Yaskawa INFORM job: OK_R2_O57-69(1)(90,0)_OK.JBI

/JOB
//NAME OK_R2_O57-69(1)(90,0)_OK
///FOLDERNAME X4
//POS
///NPOS 455,455,455,17,0,0
///TOOL 0
///POSTYPE PULSE
///PULSE
C00000=142687,-11580,-21865,-46298,77318,26406
C00001=107635,105639,59193,-4004,83878,4369
C00002=107385,112835,71659,-3962,79901,4413
C00003=107289,116273,78306,-3960,77580,4454
C00004=107289,116207,79332,-3970,76915,4475
C00005=107289,116273,78306,-3960,77580,4454
C00006=107447,123392,87902,-4042,75345,4582
C00007=107368,119615,82796,-3999,76540,4514
C00008=107503,109882,68607,-3993,80266,4441
C00009=107756,103001,56611,-4038,84116,4400
C00010=108153,102502,65455,-9976,80197,11407
C00011=107537,110693,79141,-9943,75970,11537
C00012=107296,115242,87458,-9996,73200,11681
C00013=107296,115607,88878,-10031,72523,11737
C00014=107296,115242,87458,-9996,73200,11681
C00015=106873,122679,97490,-10001,70830,11727
C00016=107051,118089,91280,-9973,72293,11668
C00017=107734,107812,76377,-9988,76211,11587
C00018=108357,99970,63216,-10030,80298,11469
C00019=111395,81814,40298,-10763,85374,12058
C00020=135939,40633,60147,-39777,44722,28223
C00021=135273,44440,65799,-40560,43252,28620
C00022=135218,49510,74479,-42532,41149,29811
C00023=135218,52739,80290,-44069,39733,30719
C00024=135218,51401,77909,-43430,40304,30344
C00025=135400,47409,73389,-42907,40927,30065
C00026=135400,49581,77316,-43951,39968,30683
C00027=135083,52398,80539,-44303,39430,30833
C00028=135400,49581,77316,-43951,39968,30683
C00029=133089,26435,31840,-33362,51762,23582
C00030=122836,-20707,-1842,-26261,58142,44331
C00031=108542,-11029,1672,-9630,61367,37079
C00032=108679,-9299,6685,-9878,59219,37321
C00033=108679,-8233,9358,-9991,58138,37420
C00034=108679,-8832,7868,-9928,58739,37363
C00035=101227,-4424,8478,6098,64645,33408
C00036=101749,-3909,10367,6019,63714,33552
C00037=99890,-2844,11238,6455,63869,32869
C00038=101954,-4018,10279,5971,63698,33629
C00039=119599,-21935,-8687,-19541,65328,41245
C00040=157787,18659,24844,-603,57771,19260
C00041=142866,15340,32539,5422,51765,13080
C00042=142866,17061,36428,5538,50265,12998
C00043=142866,16346,34832,5489,50877,13033
C00044=143013,20262,38513,5445,50617,13080
C00045=142866,16346,34832,5489,50877,13033
C00046=132913,34622,53415,24401,61187,-11407
C00047=133468,34916,53719,24326,60995,-11227
C00048=131729,29112,41902,23735,65422,-10932
C00049=97397,-56372,-66081,25937,96155,-17363
C00050=91007,-59958,-65967,24261,97668,-32617
C00051=125926,-77250,-66316,21080,81833,-36437
C00052=126284,-594,-20029,15604,88354,-35723
C00053=126284,-509,-12976,15645,84209,-36248
C00054=124802,3877,-7879,15893,83645,-36839
C00055=124802,4020,-6552,15911,82926,-36931
C00056=124802,3943,-7243,15902,83298,-36884
C00057=123270,3785,-7378,16131,83600,-37383
C00058=123399,3884,-6575,16123,83149,-37397
C00059=123813,3922,-6544,16060,83068,-37263
C00060=123399,3797,-7355,16113,83568,-37342
C00061=129363,-46213,-49135,15183,82438,-35396
C00062=131818,-93939,-91511,4308,83147,-7603
C00063=129147,-104974,-80844,-32439,31226,48978
C00064=127581,-72421,-62371,-35585,33961,68342
C00065=124664,-66928,-57448,-32966,32611,66961
C00066=123754,-63943,-53853,-32629,31684,66786
C00067=123754,-63568,-52544,-33171,31167,67071
C00068=123754,-63943,-53853,-32629,31684,66786
C00069=123639,-59018,-51277,-31710,32448,66301
C00070=123582,-56512,-49922,-31282,32817,66076
C00071=123639,-59018,-51277,-31710,32448,66301
C00072=131982,-55244,-47165,-50372,40396,73195
C00073=130304,-55630,-47379,-49442,39430,72657
C00074=124207,-63622,-54438,-32639,32305,66790
C00075=125315,-65804,-56448,-33641,32835,67317
C00076=128233,-71228,-61365,-36187,34229,68662
C00077=123372,-90110,-48954,-69127,12132,-32175
C00078=164723,-27709,-11098,-69634,69545,-47097
C00079=168592,-14054,-1264,-69323,72507,-47019
C00080=158796,970,10778,-68977,66045,-48502
C00081=178190,-60094,-55002,-67962,82251,-43615
C00082=173027,-67602,-58858,-67784,78202,-43687
C00083=169341,-70270,-58661,-67804,75132,-43553
C00084=169341,-69900,-57436,-67934,74906,-43308
C00085=169341,-70270,-58661,-67804,75132,-43553
C00086=168190,-69795,-58431,-67693,74405,-43758
C00087=166974,-69170,-58127,-67562,73648,-43988
C00088=168190,-69795,-58431,-67693,74405,-43758
C00089=173339,-68324,-59217,-67832,78352,-43578
C00090=179024,-58740,-54280,-67998,82909,-43609
C00091=180089,-62311,-56169,-68129,83355,-43176
C00092=195989,-67260,-58691,-68544,93647,-40636
C00093=215727,-82846,-65910,-66533,105415,-36335
C00094=205418,-117613,-84907,-62264,88933,-23433
C00095=200540,-66438,-67217,-63628,100285,15829
C00096=127293,-88890,-117674,-21964,112183,47373
C00097=127884,-113870,-117586,-20406,100261,49782
C00098=126455,-94233,-83658,-19548,96625,49926
C00099=122769,-95152,-80887,-19686,93685,49072
C00100=121257,-92855,-76623,-19731,91957,48808
C00101=121256,-92184,-75240,-19721,91480,48885
C00102=121257,-92855,-76623,-19731,91957,48808
C00103=119709,-92847,-76620,-19813,91585,48312
C00104=118447,-92805,-76604,-19874,91287,47906
C00105=121134,-93057,-78029,-19757,92646,48652
C00106=122616,-92853,-79205,-19699,93786,49000
C00107=126246,-91944,-81970,-19569,96706,49837
C00108=116739,-91029,-87152,11175,94833,-69838
C00109=118638,-93558,-84500,11112,91693,-69464
C00110=121559,-94813,-81066,11067,88585,-68734
C00111=121559,-94454,-79960,11067,88097,-68778
C00112=121559,-94813,-81066,11067,88585,-68734
C00113=121580,-97932,-82261,11067,87731,-68801
C00114=121559,-94813,-81066,11067,88585,-68734
C00115=124478,-94674,-81011,11026,88221,-67759
C00116=121559,-94813,-81066,11067,88585,-68734
C00117=121199,-93273,-83309,11082,90766,-68663
C00118=119237,-90980,-86060,11143,93854,-69064
C00119=119262,-91078,-98551,11400,101347,-68370
C00120=119262,-88450,-105465,11733,106843,-67839
C00121=123634,-129086,-124562,-18007,62786,21453
C00122=124713,-112307,-109989,-18584,62695,21889
C00123=121750,-102661,-104576,-16897,63614,20597
C00124=120661,-96847,-100545,-16291,63882,20142
C00125=120661,-96945,-99213,-16408,63045,20264
C00126=120661,-96847,-100545,-16291,63882,20142
C00127=119434,-96825,-100537,-15680,63651,19709
C00128=118199,-96764,-100511,-15059,63439,19270
C00129=119434,-96825,-100537,-15680,63651,19709
C00130=120468,-95018,-99831,-16130,64325,20004
C00131=120473,-92385,-98782,-16042,65005,19908
C00132=120468,-95018,-99831,-16130,64325,20004
C00133=121400,-102567,-103315,-16828,62845,20579
C00134=124338,-112119,-108698,-18515,61948,21869
C00135=115152,-110094,-108973,21966,66789,-27187
C00136=118701,-101887,-103909,20282,66922,-25804
C00137=120033,-96498,-99821,19662,66842,-25314
C00138=120033,-96571,-98630,19770,66116,-25442
C00139=120033,-96498,-99821,19662,66842,-25314
C00140=121038,-96503,-99823,19217,66607,-24975
C00141=122863,-96447,-99800,18396,66209,-24352
C00142=121038,-96503,-99823,19217,66607,-24975
C00143=121031,-93073,-98698,19079,67622,-24806
C00144=121028,-91162,-97925,19016,68103,-24728
C00145=121031,-93073,-98698,19079,67622,-24806
C00146=119849,-101075,-102503,19842,66224,-25492
C00147=116381,-109262,-107580,21511,66068,-26853
C00148=114174,-113759,-109466,25218,61256,-29915
C00149=117999,-105066,-104585,23039,61495,-28291
C00150=119436,-99712,-100384,22286,61259,-27759
C00151=119436,-99710,-99356,22420,60673,-27881
C00152=119436,-99712,-100384,22286,61259,-27759
C00153=121229,-99730,-100389,21374,60785,-27131
C00154=123455,-99637,-100354,20211,60254,-26337
C00155=121229,-99730,-100389,21374,60785,-27131
C00156=121193,-87849,-97584,20616,64895,-26352
C00157=121184,-85182,-96456,20515,65531,-26236
C00158=121193,-87849,-97584,20616,64895,-26352
C00159=119818,-94456,-100985,21520,64018,-27049
C00160=116346,-102514,-105912,23431,63914,-28430
C00161=120616,-96535,-104175,23887,64719,-45568
C00162=120616,-96992,-102054,24182,63306,-45881
C00163=136389,-91621,-102582,2930,64785,-40204
C00164=118869,-97062,-101163,25162,63282,-46587
C00165=120614,-98220,-102778,24220,63138,-45920
C00166=133621,-94767,-111832,11795,91375,-37411
C00167=135524,-95930,-105043,10399,87493,-38783
C00168=135817,-95923,-103691,10152,86855,-39072
C00169=120616,-96793,-103087,23408,87451,-42960
C00170=120617,-96070,-105685,23410,89266,-42604
C00171=120635,-118119,-124325,17957,114364,-37370
C00172=107148,-122068,-106720,37591,45003,-56343
C00173=107143,-118125,-97071,40168,41922,-57944
C00174=107140,-117153,-94914,40772,41285,-58308
C00175=108973,-111199,-92224,38587,41539,-56980
C00176=105115,-116142,-93852,42098,42144,-59139
C00177=107012,-118507,-95796,40965,41228,-58425
C00178=106841,-125065,-112650,27659,77705,-49700
C00179=108922,-124444,-112086,25532,82947,-48175
C00180=119544,-112769,-109618,11884,115103,-48129
C00181=107149,-124464,-114807,14035,115464,-42498
C00182=107153,-124980,-118069,14274,117155,-42276
C00183=120683,-72727,-118704,1403,106780,-1205
C00184=120616,-97084,-101761,-23685,56760,46645
C00185=120615,-97341,-97713,-24403,54354,47226
C00186=120615,-97245,-95574,-24781,53197,47519
C00187=114204,-97094,-94072,-16119,48782,41960
C00188=120613,-98403,-96349,-24817,53089,47545
C00189=122362,-97151,-94697,-25998,53280,48291
C00190=118994,-95787,-106265,-23004,89078,41795
C00191=118527,-107245,-109313,-22939,85243,42364
C00192=120617,-95328,-107797,-23350,90604,42068
C00193=120618,-93989,-110172,-23402,92584,41681
C00194=120619,-87370,-116055,-23793,99045,40394
C00195=120619,-87370,-116055,-23793,99045,40394
C00196=120618,-86394,-114990,8935,74593,77376
C00197=120618,-89943,-112390,9089,71210,77123
C00198=120618,-91094,-111253,9157,69935,77026
C00199=120921,-87010,-110025,8929,71231,77225
C00200=120616,-91696,-112687,9127,70502,77069
C00201=120617,-91433,-110915,9280,69085,76949
C00202=120617,-91707,-110620,9342,68290,76888
C00203=120617,-92092,-110153,9289,66860,76810
C00204=120617,-92703,-109346,8604,64312,76688
C00205=120617,-93084,-108807,7222,62458,76641
C00206=120617,-93193,-108666,5837,61715,76664
C00207=120618,-90875,-111661,5103,64613,76670
C00208=120618,-90809,-111742,4197,64653,76687
C00209=120618,-90545,-112027,2634,65244,76730
C00210=120618,-90001,-112556,1051,66686,76779
C00211=120618,-89211,-113241,-130,68806,76818
C00212=120618,-88484,-113805,-667,70701,76840
C00213=120618,-87123,-114601,-725,72803,76709
C00214=120619,-86169,-115177,-666,75079,76754
C00215=120619,-85009,-115798,44,77805,76866
C00216=120619,-84186,-116189,1368,79788,77043
C00217=120619,-83945,-116287,2643,80551,77203
C00218=118270,-87908,-113898,4548,77310,76315
C00219=117006,-87882,-113777,5977,77383,75992
C00220=115001,-87936,-113393,8376,77055,75464
C00221=113157,-88199,-112730,10795,75966,74930
C00222=112003,-88721,-111920,12625,74164,74513
C00223=111959,-89151,-111512,13141,72976,74431
C00224=114352,-90005,-111461,12180,71784,75105
C00225=117604,-90791,-111341,10710,70486,76060
C00226=117404,-89600,-112462,10735,71791,76111
C00227=116906,-85938,-115017,10812,75246,76259
C00228=120614,-97623,-100799,20300,88883,-51757
C00229=120614,-96302,-87355,20440,81742,-52958
C00230=120613,-95405,-83784,20521,80111,-53236
C00231=126109,-109592,-85843,18017,65653,-40663
C00232=119108,-93712,-82042,20736,80300,-53753
C00233=120703,-96440,-84059,20528,79748,-53266
C00234=121011,-95101,-82657,16234,85393,-56932
C00235=120815,-94676,-79544,16280,83804,-57215
C00236=120149,-97496,-80464,13581,88226,-67082
C00237=120613,-95181,-82964,13310,91650,-67966
C00238=120614,-96223,-86939,13345,93512,-67766
C00239=120615,-97634,-95801,13498,98116,-67263
C00240=121294,-114205,-91205,-24827,58618,34956
C00241=120612,-94063,-79189,-30374,49118,27390
C00242=120612,-92317,-74276,-31337,47279,28045
C00243=120611,-91635,-72532,-31685,46659,28276
C00244=118073,-86207,-69815,-27979,45725,25770
C00245=120609,-92794,-73597,-31655,46709,28256
C00246=122365,-91337,-71823,-32796,47086,29053
C00247=115372,-110415,-90260,-20403,67055,37755
C00248=116442,-100471,-77078,-21305,66259,40654
C00249=116372,-94168,-76064,-20320,81539,56413
C00250=120612,-93792,-78416,-23522,88402,60481
C00251=120613,-94966,-82014,-23532,89885,60189
C00252=192979,-49879,-84133,-31949,90821,59300
C00253=226136,-49296,-77583,-43048,96139,60221
C00254=194231,-43574,-37464,-64429,96533,-35524
C00255=168190,-921,2356,-69742,86936,-65420
C00256=167171,-9679,-4727,-69794,80481,-66551
C00257=161668,-12899,-4972,-71887,72051,-48991
C00258=158364,-12022,-5998,-68672,69294,-39906
C00259=156881,-17849,-10944,-69825,79076,-66625
C00260=156054,-17027,-11609,-69675,78824,-67093
C00261=158331,-12175,-6115,-68672,69269,-39907
C00262=156361,-14598,-7677,-68484,66767,-40276
C00263=151900,-18330,-10475,-67308,59054,-41902
C00264=154261,3537,6976,-69079,75732,-38618
C00265=154747,-10639,-6391,-66828,75297,-54318
C00266=154442,-11587,-10980,-61883,80878,-64503
C00267=159305,-13086,-7363,-68622,70046,-39902
C00268=160610,-11568,-6196,-68690,70948,-39749
C00269=179726,-19719,-12316,-69264,83687,-37039
C00270=180202,-65513,-36112,-70171,79517,-38597
C00271=171321,-47804,-23743,-70196,73038,-45095
C00272=120855,-117042,-83065,-287,50429,281
C00273=120852,-56541,-79529,-233,79340,219
C00274=120696,53119,40617,-185,61751,192
C00275=120686,117420,104140,-194,55702,198
C00276=120685,99043,82380,-184,59649,191
C00277=122493,102932,90070,-987,56926,916
C00278=120685,123863,115449,-202,52052,205
C00279=120704,115543,105340,-205,53998,209
C00280=122467,102927,90062,-975,56928,906
C00281=121054,101096,87697,-350,57430,341
C00282=121218,100526,86952,-2924,57717,2680
C00283=119871,97554,82980,-2313,58589,2128
C00284=121770,99804,85898,-7979,58802,7335
C00285=123458,93230,74100,-8365,62819,7694
C00286=127901,89142,85055,-16058,61001,15638
C00287=140740,128608,122591,-17053,51761,14935
C00288=141173,120915,113217,-16837,53591,14809
C00289=125539,79311,72650,-14999,63041,14428
C00290=124982,76834,69616,-14757,63515,14150
C00291=126480,71694,61185,-14909,66256,14364
C00292=127425,72489,65068,-16510,65063,16091
C00293=151716,35869,40711,-43800,85634,42977
C00294=153219,23704,46468,-39932,89274,45297
C00295=150010,47902,71614,-40707,85512,45394
C00296=154240,23283,29848,-40334,97498,42612
C00297=154465,34676,28167,-3963,80968,257
C00298=157399,18456,15561,6305,73633,-11364
C00299=166913,17393,14571,4349,73064,-8034
C00300=170742,26415,26762,1268,69531,-3078
C00301=170212,26486,27746,1388,68971,-3275
C00302=169116,27159,30341,1645,67741,-3687
C00303=176334,39723,42022,-11916,74582,1979
C00304=182119,52793,59875,-23973,76306,25334
C00305=185046,47030,49277,-23757,80416,25586
C00306=156159,-27844,-33931,-20967,84276,14245
C00307=135002,-107739,-89418,-17788,72722,8424
C00308=182779,-47107,-63468,-4299,76483,-82831
C00309=189334,-126614,-108463,-44477,62316,-64668
C00310=121693,-126430,-88761,-53982,17457,-73114
C00311=140282,-82155,-73154,-59383,46557,-69401
C00312=137402,-83281,-73645,-58395,44635,-69973
C00313=132931,-76557,-73113,-49425,46479,-74892
C00314=136898,-85885,-74084,-59112,43749,-69513
C00315=136236,-83853,-74475,-57682,44042,-70397
C00316=132981,-76543,-73106,-49450,46508,-74878
C00317=119425,-90003,-77331,-28870,26914,-75911
C00318=135712,-71182,-68173,-46953,38713,-58640
C00319=143905,-59721,-61352,-57730,51418,-39205
C00320=121775,-86236,-74909,-25532,24619,-52498
C00321=121774,-86244,-74912,-25532,24617,-52498
C00322=121693,-126430,-88761,-53982,17457,-73114
C00323=118534,-85327,-101542,31688,82312,-3081
C00324=113867,24354,-27186,33136,92965,-1727
C00325=160796,40344,30640,17217,54638,7315
C00326=160797,40341,30637,17217,54638,7315
C00327=160797,40341,30637,17217,54638,7315
C00328=160252,39151,28676,17378,55324,7200
C00329=161178,38223,28434,16963,54814,7508
C00330=160796,40350,30646,17218,54637,7315
C00331=160795,40351,30648,17218,54637,7314
C00332=160794,40354,30651,17218,54637,7314
C00333=134054,6396,-12292,27269,70214,-305
C00334=134055,6392,-12295,27269,70214,-305
C00335=134055,6392,-12295,27269,70214,-305
C00336=133335,6117,-13247,27465,70843,-432
C00337=134208,4264,-14132,27207,70198,-248
C00338=134055,6400,-12288,27269,70214,-305
C00339=134054,6402,-12286,27269,70214,-305
C00340=134054,6405,-12283,27270,70214,-305
C00341=134054,6378,-12307,27269,70215,-305
C00342=110297,92470,61471,162,75039,5870
C00343=106536,92878,46535,-6489,85409,6991
C00344=105889,102407,60005,-6334,81981,6955
C00345=107411,109724,75819,-6896,76174,7779
C00346=107307,113841,80039,-6878,75687,7770
C00347=106147,102899,60646,-6410,81858,7045
C00348=107454,121313,92229,795,70933,3205
C00349=107823,121162,91899,673,71054,3335
C00350=103297,112702,80407,10779,76295,-8281
C00351=100760,114985,83493,16597,79533,-16127
C00352=102994,101893,66401,15964,82735,-14918
C00353=102438,121053,88749,15854,82872,-18908
C00354=103348,86539,46576,12183,80201,-18226
C00355=107306,113906,81371,827,73803,3171
C00356=107311,117545,72428,-13995,85411,11857
C00357=105409,119135,76795,-9100,84379,11874
C00358=104759,108123,65686,-7737,79041,12181
C00359=107310,116811,74228,-14018,83968,12019
C00360=107566,113040,70432,-14074,84397,12057
C00361=105955,98232,55061,-11625,77681,12450
C00362=106075,100097,56813,-12565,79285,12270
C00363=104774,97118,52951,-12100,79924,11770
C00364=104167,97049,52732,-11892,79935,11566
C00365=103488,98146,54277,-11675,79461,11386
C00366=105019,93844,46472,-12276,82982,11528
C00367=107312,117616,72525,-13996,85389,11860
C00368=113054,94415,53645,-15341,86201,13636
C00369=132655,10139,3212,-19793,78564,21692
C00370=120395,-86682,-93138,-17072,84894,16376
C00371=120731,-81008,-115648,105,86416,81801
C00372=120675,-24654,-47163,132,73228,81771
C00373=120676,-24640,-47153,131,73229,81771
C00374=121102,-22780,-44290,-48,72423,81914
C00375=120676,-24370,-48215,131,74021,81772
C00376=121750,-24626,-47144,-317,73232,82133
C00377=121088,-18910,-41523,-41,72708,81911
C00378=120676,-24640,-47153,131,73229,81771
C00379=120672,-32524,-49889,133,70864,81769
C00380=86683,-40445,-63075,13763,77736,70672
C00381=103499,26970,-9106,7161,77072,76192
C00382=140778,108078,66600,20509,92089,48724
C00383=140778,108101,66629,20508,92083,48723
C00384=140777,108123,66659,20508,92077,48722
C00385=140791,110557,71328,20474,90549,48468
C00386=140777,108420,65802,20527,92715,48830
C00387=141368,109052,67884,20414,91674,48860
C00388=140538,117676,80864,20492,88534,48038
C00389=140777,108123,66659,20508,92077,48722
C00390=140778,108101,66629,20508,92083,48723
C00391=140778,108101,66629,20508,92083,48723
C00392=140778,108122,66658,20508,92077,48722
C00393=140768,108703,68758,20489,91145,48562
C00394=140777,108420,65801,20527,92715,48830
C00395=141368,109051,67883,20414,91674,48860
C00396=140511,115176,77354,20500,89363,48171
C00397=140778,108122,66658,20508,92077,48722
C00398=140778,108100,66628,20508,92083,48723
C00399=140778,108078,66599,20509,92089,48724
C00400=126581,14025,-47477,25241,115824,48542
C00401=159492,92702,46653,29136,105568,44545
C00402=162149,88036,41181,28914,105145,45798
C00403=163325,88052,47564,28312,101300,45262
C00404=160866,111719,71725,28335,100123,43674
C00405=160864,108336,66000,28535,101703,44070
C00406=164354,88224,47874,28236,100875,45547
C00407=160866,108108,66623,28476,101259,43959
C00408=161429,110004,69125,28389,100573,44000
C00409=160867,107600,68720,43807,97992,44930
C00410=160869,107245,72152,43546,96305,44200
C00411=160853,112270,81548,43267,93953,43186
C00412=160872,111361,79145,43345,94689,43509
C00413=160869,107230,72446,43527,96165,44140
C00414=161852,112523,81931,43214,93388,43402
C00415=160870,107231,72133,43547,96307,44201
C00416=160868,107586,68702,43807,97995,44932
C00417=160873,107541,68625,43810,98010,44941
C00418=160875,107181,72050,43549,96324,44211
C00419=160969,112164,81513,43259,93871,43205
C00420=160878,111286,79028,43348,94711,43521
C00421=160875,107165,72344,43530,96184,44151
C00422=161946,112277,81723,43208,93342,43426
C00423=160876,107167,72031,43549,96326,44212
C00424=160874,107528,68607,43810,98012,44942
C00425=160865,108116,66633,19225,80466,-79641
C00426=160864,108012,67019,19239,80191,-79685
C00427=160902,111102,73963,19378,77641,-80084
C00428=160868,111461,73140,19346,78303,-79987
C00429=160865,107941,67240,19247,80028,-79711
C00430=161896,111383,74336,19093,77331,-79779
C00431=160866,107998,67001,19238,80195,-79684
C00432=160866,108102,66615,19224,80470,-79640
C00433=141960,25007,-13534,18907,77065,-75548
C00434=148396,38776,-224,4331,80270,-75408
C00435=147937,42862,4060,4507,79758,-75574
C00436=147586,38479,-2882,4613,81790,-75612
C00437=132676,28155,-16568,22865,92034,-69453
C00438=139622,-24488,-52979,20482,85647,-66084
C00439=105595,-117820,-100492,25848,75539,-72989
C00440=106580,-108863,-97500,25415,77736,-72126
C00441=109054,-118504,-91401,16987,64899,-66879
C00442=114351,-116427,-87550,15194,62531,-65147
C00443=119485,-94955,-76898,12502,65960,-62737
C00444=99170,-109633,-81201,29999,68590,-70531
C00445=97263,-108225,-79726,30318,69111,-71170
C00446=119688,-71486,-66798,11989,71648,-62069
C00447=119489,-72073,-70371,11931,73536,-61952
C00448=119715,-43131,-54580,11630,78554,-61387
C00449=119934,-43288,-51446,11646,76556,-61502
C00450=120006,-17553,-34071,11532,79027,-61243
C00451=119832,-16968,-37707,11506,81540,-61066
C00452=138269,-21321,-44343,-15851,46320,-74175
C00453=176671,-154466,-104215,-64912,39697,-45563
C00454=34524,-124554,-102946,-40349,70974,-61921
BC00000=343252,458654,396766
BC00001=296461,362277,161319
BC00002=296461,362277,161319
BC00003=296461,362277,161318
BC00004=296461,362277,161318
BC00005=296461,362277,161318
BC00006=296461,362277,161318
BC00007=296461,362277,161318
BC00008=296461,362277,161319
BC00009=296461,362277,161319
BC00010=305664,365412,228193
BC00011=305664,365412,228193
BC00012=305664,365412,228193
BC00013=305664,365412,228193
BC00014=305664,365412,228193
BC00015=305664,365412,228193
BC00016=305664,365412,228193
BC00017=305664,365412,228193
BC00018=305664,365412,228193
BC00019=305664,365412,228193
BC00020=308753,366328,364268
BC00021=308753,366328,364268
BC00022=308753,366328,364268
BC00023=308753,366328,364268
BC00024=308753,366328,364268
BC00025=308753,366328,364268
BC00026=308753,366328,364268
BC00027=308753,366328,364268
BC00028=308753,366328,364268
BC00029=301860,366328,381931
BC00030=269052,381689,418036
BC00031=269052,381689,418036
BC00032=269052,381689,418036
BC00033=269052,381689,418036
BC00034=269052,381689,418036
BC00035=269052,381689,418036
BC00036=269052,381689,418036
BC00037=269052,381689,418036
BC00038=269052,381689,418036
BC00039=269052,381689,418036
BC00040=313126,381689,418036
BC00041=269052,381689,418036
BC00042=269052,381689,418036
BC00043=269052,381689,418036
BC00044=269052,381689,418036
BC00045=269052,381689,418036
BC00046=269052,381689,418036
BC00047=269052,381689,418036
BC00048=269052,381689,418036
BC00049=269052,381689,467818
BC00050=289570,498982,521007
BC00051=178478,467489,256734
BC00052=178478,467489,256734
BC00053=178478,467489,256734
BC00054=178478,467489,256734
BC00055=178478,467489,256734
BC00056=178478,467489,256734
BC00057=178478,467489,256734
BC00058=178478,467489,256734
BC00059=178478,467489,256734
BC00060=178478,467489,256734
BC00061=178478,467489,256734
BC00062=138740,481045,202237
BC00063=61948,507240,96923
BC00064=3185,506590,90506
BC00065=1592,506590,90506
BC00066=1592,506590,90506
BC00067=1592,506590,90506
BC00068=1592,506590,90506
BC00069=1592,506590,90506
BC00070=1592,506590,90506
BC00071=1592,506590,90506
BC00072=1592,506590,90506
BC00073=1592,506590,90506
BC00074=1592,506590,90506
BC00075=1592,506590,90506
BC00076=1592,506590,90506
BC00077=2850,506353,232671
BC00078=1592,518884,229372
BC00079=1592,518884,229372
BC00080=1593,518883,229370
BC00081=1592,449343,97956
BC00082=1592,445130,78954
BC00083=1592,443444,71348
BC00084=1592,443444,71348
BC00085=1592,443444,71348
BC00086=1592,443444,71348
BC00087=1592,443444,71348
BC00088=1592,443444,71348
BC00089=1592,446018,71478
BC00090=1592,450231,90479
BC00091=3185,450231,90479
BC00092=3185,450231,90479
BC00093=3185,450231,90479
BC00094=7707,456386,217176
BC00095=80806,494061,563567
BC00096=35141,510033,1075139
BC00097=35141,419749,1075139
BC00098=34345,418785,1075139
BC00099=34345,418785,1075139
BC00100=34345,418785,1075139
BC00101=34345,418785,1075139
BC00102=34345,418785,1075139
BC00103=34345,418785,1075139
BC00104=34345,418785,1075139
BC00105=34345,418785,1075139
BC00106=34345,418785,1075139
BC00107=34345,418785,1075139
BC00108=42781,423417,1075139
BC00109=42781,423417,1075139
BC00110=42781,423417,1075139
BC00111=42781,423417,1075139
BC00112=42781,423417,1075139
BC00113=42781,423417,1075139
BC00114=42781,423417,1075139
BC00115=42781,423417,1075139
BC00116=42781,423417,1075139
BC00117=42781,423417,1075139
BC00118=42781,423417,1075139
BC00119=42781,423417,1075139
BC00120=42781,423417,1075139
BC00121=146006,330330,1075139
BC00122=146006,330330,1075139
BC00123=146006,330330,1075139
BC00124=146006,330330,1075139
BC00125=146006,330330,1075139
BC00126=146006,330330,1075139
BC00127=146006,330330,1075139
BC00128=146006,330330,1075139
BC00129=146006,330330,1075139
BC00130=146006,330330,1075139
BC00131=146006,330330,1075139
BC00132=146006,330330,1075139
BC00133=146006,330330,1075139
BC00134=146006,330330,1075139
BC00135=176033,332548,1075139
BC00136=176033,332548,1075139
BC00137=176033,332548,1075139
BC00138=176033,332548,1075139
BC00139=176033,332548,1075139
BC00140=176033,332548,1075139
BC00141=176033,332548,1075139
BC00142=176033,332548,1075139
BC00143=176033,332548,1075139
BC00144=176033,332548,1075139
BC00145=176033,332548,1075139
BC00146=176033,332548,1075139
BC00147=176033,332548,1075139
BC00148=129718,348283,1075139
BC00149=129718,348283,1075139
BC00150=129718,348283,1075139
BC00151=129718,348283,1075139
BC00152=129718,348283,1075139
BC00153=129718,348283,1075139
BC00154=129718,348283,1075139
BC00155=129718,348283,1075139
BC00156=129718,348283,1075139
BC00157=129718,348283,1075139
BC00158=129718,348283,1075139
BC00159=129718,348283,1075139
BC00160=129718,348283,1075139
BC00161=142137,344452,1075139
BC00162=136685,340806,1075139
BC00163=134504,339347,1075139
BC00164=134504,339347,1075139
BC00165=134504,339347,1075139
BC00166=137500,303887,1075136
BC00167=137704,341068,1075138
BC00168=137746,348694,1075139
BC00169=139991,349177,1075139
BC00170=145603,350382,1075139
BC00171=180440,260677,1075139
BC00172=168005,343926,1075139
BC00173=168026,343923,1075139
BC00174=162990,339007,1075139
BC00175=160976,337041,1075139
BC00176=160976,337041,1075139
BC00177=160976,337041,1075139
BC00178=169541,293251,1075139
BC00179=171223,294834,1075136
BC00180=160286,251960,1075135
BC00181=160091,242762,1075139
BC00182=164957,240749,1075139
BC00183=157878,329403,1075139
BC00184=127205,341832,1075139
BC00185=127216,341831,1075139
BC00186=132492,337593,1075139
BC00187=134583,335912,1075135
BC00188=134603,335898,1075139
BC00189=134603,335898,1075139
BC00190=128692,290623,1075139
BC00191=128692,290623,1075139
BC00192=126432,295463,1075139
BC00193=120824,296710,1075139
BC00194=120803,296713,1075139
BC00195=108643,383849,1075139
BC00196=397017,323220,1075139
BC00197=396327,320708,1075139
BC00198=396051,319704,1075139
BC00199=396051,319704,1075139
BC00200=396051,319704,1075139
BC00201=391487,321222,1075139
BC00202=388835,322408,1075139
BC00203=387826,323910,1075139
BC00204=385565,326420,1075139
BC00205=382298,328058,1075139
BC00206=379434,328404,1075139
BC00207=374349,308859,1075139
BC00208=372612,308545,1075139
BC00209=369837,307583,1075139
BC00210=367229,305822,1075139
BC00211=365511,303458,1075139
BC00212=365104,301418,1075139
BC00213=386881,296395,1075139
BC00214=387751,294116,1075139
BC00215=389873,291541,1075139
BC00216=393077,289829,1075139
BC00217=395936,289453,1075139
BC00218=398158,308931,1075139
BC00219=398158,309255,1075139
BC00220=398158,310269,1075139
BC00221=398158,312120,1075139
BC00222=398158,314574,1075139
BC00223=398158,316012,1075139
BC00224=398158,317233,1075139
BC00225=398158,318652,1075139
BC00226=398158,319656,1075139
BC00227=398158,322168,1075139
BC00228=52314,423180,1075139
BC00229=52314,423180,1075139
BC00230=47244,423170,1075139
BC00231=45216,423166,1075139
BC00232=45216,423166,1075139
BC00233=45216,423166,1075139
BC00234=39653,414730,1075139
BC00235=48595,428988,1075139
BC00236=43751,420053,1075139
BC00237=44320,417752,1075139
BC00238=47425,415104,1075139
BC00239=47404,415107,1075139
BC00240=32765,406492,1075139
BC00241=26155,443193,1075139
BC00242=26165,443191,1075139
BC00243=30757,437510,1075139
BC00244=32593,435238,1075139
BC00245=32593,435238,1075139
BC00246=32593,435238,1075139
BC00247=29497,393908,1075139
BC00248=29640,444611,1075139
BC00249=30720,431633,1075139
BC00250=29609,420698,1075139
BC00251=24721,418722,1075139
BC00252=181425,467724,1075139
BC00253=206351,494131,993943
BC00254=43495,490453,343014
BC00255=795,489471,169163
BC00256=795,489616,176646
BC00257=795,487501,172010
BC00258=796,486242,169247
BC00259=795,487347,156245
BC00260=795,487347,156245
BC00261=796,486242,169247
BC00262=795,490466,169240
BC00263=795,499607,169190
BC00264=795,503780,169165
BC00265=795,491703,166651
BC00266=795,483818,165013
BC00267=795,487979,176733
BC00268=795,492323,195444
BC00269=795,492323,195444
BC00270=795,486278,213645
BC00271=795,493274,229372
BC00272=302356,491157,498290
BC00273=302356,472251,354240
BC00274=302356,439893,260644
BC00275=305516,442484,107552
BC00276=305553,428260,107552
BC00277=305567,425083,107552
BC00278=305568,434078,107552
BC00279=305568,434078,107552
BC00280=305567,425083,107552
BC00281=305568,424826,107552
BC00282=305568,424826,107552
BC00283=305568,424826,107552
BC00284=305568,424826,107552
BC00285=305568,424826,107552
BC00286=305568,396001,205574
BC00287=375120,424070,107552
BC00288=375120,424070,107552
BC00289=305568,396001,205574
BC00290=305568,396001,205574
BC00291=305568,396001,205574
BC00292=306263,397023,277378
BC00293=327342,410263,352342
BC00294=327795,376287,384331
BC00295=327795,376287,384331
BC00296=327795,376287,384331
BC00297=340045,385683,420309
BC00298=343044,364755,405263
BC00299=343044,346163,349622
BC00300=343090,347045,345716
BC00301=343090,347045,345716
BC00302=343090,347045,345716
BC00303=343090,347045,345716
BC00304=343090,347045,345716
BC00305=343090,347045,345716
BC00306=332717,386671,419596
BC00307=335871,487887,419596
BC00308=390657,494896,215064
BC00309=230257,475363,68296
BC00310=1592,487362,11975
BC00311=1592,488154,18507
BC00312=1592,483770,2208
BC00313=1592,482430,553
BC00314=1592,482016,17
BC00315=1592,482016,17
BC00316=1592,482430,553
BC00317=1592,482041,72
BC00318=15514,493883,17
BC00319=2874,490153,17
BC00320=1624,492089,1241
BC00321=2343,498161,17526
BC00322=1592,487362,11975
BC00323=297934,489847,452418
BC00324=297934,451559,452418
BC00325=369477,494618,225101
BC00326=365709,489278,210559
BC00327=364202,487141,204742
BC00328=364202,487141,204742
BC00329=364202,487141,204742
BC00330=365992,487133,196103
BC00331=367499,489270,201920
BC00332=371267,494610,216463
BC00333=284963,453835,157880
BC00334=281195,448495,143338
BC00335=279688,446358,137521
BC00336=279688,446358,137521
BC00337=279688,446358,137521
BC00338=281450,446351,129016
BC00339=282957,448487,134833
BC00340=286725,453828,149375
BC00341=286704,453830,203143
BC00342=296332,391084,250132
BC00343=298513,354548,182531
BC00344=299534,352709,153581
BC00345=299534,361295,198154
BC00346=299534,361295,198154
BC00347=299534,352709,153581
BC00348=302481,362088,197934
BC00349=297981,360539,197924
BC00350=297981,352834,197924
BC00351=297981,348368,197924
BC00352=297981,348368,197924
BC00353=297981,360539,197924
BC00354=297963,360615,198193
BC00355=296238,367991,224410
BC00356=285978,361278,134879
BC00357=289750,357215,134435
BC00358=289750,357214,134433
BC00359=291259,355590,134435
BC00360=291259,355590,134435
BC00361=293172,357786,134434
BC00362=301210,361949,134435
BC00363=301210,361949,134435
BC00364=301210,361949,134435
BC00365=301210,361949,134435
BC00366=301501,362441,134435
BC00367=299908,370190,134822
BC00368=301033,369213,212215
BC00369=304873,365876,472218
BC00370=304873,490004,305428
BC00371=83759,490744,9500
BC00372=83762,500251,175391
BC00373=83753,498910,148921
BC00374=83750,498374,138333
BC00375=83750,498374,138333
BC00376=83750,498374,138333
BC00377=83750,498374,138333
BC00378=83741,495303,148933
BC00379=83750,496645,175404
BC00380=83747,452762,138074
BC00381=83747,452762,138074
BC00382=197013,452967,72700
BC00383=197023,452966,45816
BC00384=197017,452289,19037
BC00385=197014,452018,8325
BC00386=197014,452018,8325
BC00387=197014,452018,8325
BC00388=197014,452018,8325
BC00389=197005,448678,19049
BC00390=197011,449355,45828
BC00391=196891,413434,45952
BC00392=196884,412757,19173
BC00393=196878,411430,8466
BC00394=196882,412486,8462
BC00395=196882,412486,8462
BC00396=196878,411430,8466
BC00397=196873,409173,19186
BC00398=196879,409850,45965
BC00399=196869,409851,72849
BC00400=171369,415032,62137
BC00401=212198,465997,35413
BC00402=211090,448808,33245
BC00403=211090,448808,33245
BC00404=211352,466457,17
BC00405=211352,466457,17
BC00406=211090,448808,33245
BC00407=208340,468151,8632
BC00408=223852,467893,29613
BC00409=206213,469334,17
BC00410=203854,470648,17
BC00411=202394,471461,16
BC00412=202910,471173,17
BC00413=202910,471173,17
BC00414=202394,471461,16
BC00415=200577,472486,17
BC00416=202935,471172,17
BC00417=191769,445272,17
BC00418=189410,446585,17
BC00419=188171,447276,15
BC00420=188466,447111,17
BC00421=188466,447111,17
BC00422=188171,447276,15
BC00423=186193,448390,17
BC00424=188551,447076,17
BC00425=212575,472931,21903
BC00426=210217,474245,17
BC00427=209273,474770,17
BC00428=209273,474770,17
BC00429=209273,474770,17
BC00430=209273,474770,17
BC00431=206940,476083,17
BC00432=209298,474769,21903
BC00433=192891,468327,82761
BC00434=192891,468327,82761
BC00435=192891,468327,82761
BC00436=192891,468327,82761
BC00437=184343,464971,114468
BC00438=179771,447734,125423
BC00439=167626,451235,171835
BC00440=167626,424773,159262
BC00441=157596,400654,186139
BC00442=157596,400654,186139
BC00443=157596,400654,186139
BC00444=157596,400654,186139
BC00445=157596,400654,186139
BC00446=157596,400654,186139
BC00447=157596,400654,186139
BC00448=157596,400654,186139
BC00449=157596,400654,186139
BC00450=157596,400654,186139
BC00451=157596,400654,186139
BC00452=164097,426729,121152
BC00453=164097,478377,121152
BC00454=279709,491733,1053139
EC00000=-798156,-183832
EC00001=-798156,-183832
EC00002=-798156,-183832
EC00003=-798156,-183832
EC00004=-798156,-183832
EC00005=-798156,-183832
EC00006=-798156,-183832
EC00007=-798156,-183832
EC00008=-798156,-183832
EC00009=-798156,-183832
EC00010=-798156,-183832
EC00011=-798156,-183832
EC00012=-798156,-183832
EC00013=-798156,-183832
EC00014=-798156,-183832
EC00015=-798156,-183832
EC00016=-798156,-183832
EC00017=-798156,-183832
EC00018=-798156,-183832
EC00019=-798156,-183832
EC00020=-798156,-183832
EC00021=-798156,-183832
EC00022=-798156,-183832
EC00023=-798156,-183832
EC00024=-798156,-183832
EC00025=-798156,-183832
EC00026=-798156,-183832
EC00027=-798156,-183832
EC00028=-798156,-183832
EC00029=-798156,-183832
EC00030=-798156,-183832
EC00031=-798156,-183832
EC00032=-798156,-183832
EC00033=-798156,-183832
EC00034=-798156,-183832
EC00035=-798156,-183832
EC00036=-798156,-183832
EC00037=-798156,-183832
EC00038=-798156,-183832
EC00039=-798156,-183832
EC00040=-798156,-183832
EC00041=-798156,-183832
EC00042=-798156,-183832
EC00043=-798156,-183832
EC00044=-798156,-183832
EC00045=-798156,-183832
EC00046=-798156,-183832
EC00047=-798156,-183832
EC00048=-798156,-183832
EC00049=-798156,-183832
EC00050=-798156,-183832
EC00051=-798156,-183832
EC00052=-798156,-183832
EC00053=-798156,-183832
EC00054=-798156,-183832
EC00055=-798156,-183832
EC00056=-798156,-183832
EC00057=-798156,-183832
EC00058=-798156,-183832
EC00059=-798156,-183832
EC00060=-798156,-183832
EC00061=-798156,-183832
EC00062=-798156,-183832
EC00063=-798156,-183832
EC00064=-798156,-183832
EC00065=-798156,-183832
EC00066=-798156,-183832
EC00067=-798156,-183832
EC00068=-798156,-183832
EC00069=-798156,-183832
EC00070=-798156,-183832
EC00071=-798156,-183832
EC00072=-798156,-183832
EC00073=-798156,-183832
EC00074=-798156,-183832
EC00075=-798156,-183832
EC00076=-798156,-183832
EC00077=-798156,-183832
EC00078=-798156,-183832
EC00079=-798156,-183832
EC00080=-798154,-183832
EC00081=-798156,-183832
EC00082=-798156,-183832
EC00083=-798156,-183832
EC00084=-798156,-183832
EC00085=-798156,-183832
EC00086=-798156,-183832
EC00087=-798156,-183832
EC00088=-798156,-183832
EC00089=-798156,-183832
EC00090=-798156,-183832
EC00091=-798156,-183832
EC00092=-798156,-183832
EC00093=-798156,-183832
EC00094=-820978,-183832
EC00095=-883374,-183832
EC00096=-975524,-183832
EC00097=-975524,-183832
EC00098=-975524,-183832
EC00099=-975524,-183832
EC00100=-975524,-183832
EC00101=-975524,-183832
EC00102=-975524,-183832
EC00103=-975524,-183832
EC00104=-975524,-183832
EC00105=-975524,-183832
EC00106=-975524,-183832
EC00107=-975524,-183832
EC00108=-975524,-183832
EC00109=-975524,-183832
EC00110=-975524,-183832
EC00111=-975524,-183832
EC00112=-975524,-183832
EC00113=-975524,-183832
EC00114=-975524,-183832
EC00115=-975524,-183832
EC00116=-975524,-183832
EC00117=-975524,-183832
EC00118=-975524,-183832
EC00119=-975524,-183832
EC00120=-975524,-183832
EC00121=-975524,-183832
EC00122=-975524,-183832
EC00123=-975524,-183832
EC00124=-975524,-183832
EC00125=-975524,-183832
EC00126=-975524,-183832
EC00127=-975524,-183832
EC00128=-975524,-183832
EC00129=-975524,-183832
EC00130=-975524,-183832
EC00131=-975524,-183832
EC00132=-975524,-183832
EC00133=-975524,-183832
EC00134=-975524,-183832
EC00135=-975524,-183832
EC00136=-975524,-183832
EC00137=-975524,-183832
EC00138=-975524,-183832
EC00139=-975524,-183832
EC00140=-975524,-183832
EC00141=-975524,-183832
EC00142=-975524,-183832
EC00143=-975524,-183832
EC00144=-975524,-183832
EC00145=-975524,-183832
EC00146=-975524,-183832
EC00147=-975524,-183832
EC00148=-975524,-183832
EC00149=-975524,-183832
EC00150=-975524,-183832
EC00151=-975524,-183832
EC00152=-975524,-183832
EC00153=-975524,-183832
EC00154=-975524,-183832
EC00155=-975524,-183832
EC00156=-975524,-183832
EC00157=-975524,-183832
EC00158=-975524,-183832
EC00159=-975524,-183832
EC00160=-975524,-183832
EC00161=-975524,-183832
EC00162=-975524,-183832
EC00163=-975524,-183832
EC00164=-975524,-183832
EC00165=-975524,-183832
EC00166=-975521,-183833
EC00167=-975523,-183832
EC00168=-975524,-183832
EC00169=-975524,-183832
EC00170=-975524,-183832
EC00171=-975524,-183832
EC00172=-975524,-183832
EC00173=-975524,-183832
EC00174=-975524,-183832
EC00175=-975524,-183832
EC00176=-975524,-183832
EC00177=-975524,-183832
EC00178=-975524,-183832
EC00179=-975521,-183833
EC00180=-975522,-183832
EC00181=-975524,-183832
EC00182=-975524,-183832
EC00183=-975524,-183832
EC00184=-975524,-183832
EC00185=-975524,-183832
EC00186=-975524,-183832
EC00187=-975521,-183832
EC00188=-975524,-183832
EC00189=-975524,-183832
EC00190=-975524,-183832
EC00191=-975524,-183832
EC00192=-975524,-183832
EC00193=-975524,-183832
EC00194=-975524,-183832
EC00195=-975524,-183832
EC00196=-975524,-183832
EC00197=-975524,-183832
EC00198=-975524,-183832
EC00199=-975524,-183832
EC00200=-975524,-183832
EC00201=-975524,-183832
EC00202=-975524,-183832
EC00203=-975524,-183832
EC00204=-975524,-183832
EC00205=-975524,-183832
EC00206=-975524,-183832
EC00207=-975524,-183832
EC00208=-975524,-183832
EC00209=-975524,-183832
EC00210=-975524,-183832
EC00211=-975524,-183832
EC00212=-975524,-183832
EC00213=-975524,-183832
EC00214=-975524,-183832
EC00215=-975524,-183832
EC00216=-975524,-183832
EC00217=-975524,-183832
EC00218=-975524,-183832
EC00219=-975524,-183832
EC00220=-975524,-183832
EC00221=-975524,-183832
EC00222=-975524,-183832
EC00223=-975524,-183832
EC00224=-975524,-183832
EC00225=-975524,-183832
EC00226=-975524,-183832
EC00227=-975524,-183832
EC00228=-975524,-183832
EC00229=-975524,-183832
EC00230=-975524,-183832
EC00231=-975524,-183832
EC00232=-975524,-183832
EC00233=-975524,-183832
EC00234=-975524,-183832
EC00235=-975524,-183832
EC00236=-975524,-183832
EC00237=-975524,-183832
EC00238=-975524,-183832
EC00239=-975524,-183832
EC00240=-975524,-183832
EC00241=-975524,-183832
EC00242=-975524,-183832
EC00243=-975524,-183832
EC00244=-975524,-183832
EC00245=-975524,-183832
EC00246=-975524,-183832
EC00247=-975524,-183832
EC00248=-975524,-183832
EC00249=-975524,-183832
EC00250=-975524,-183832
EC00251=-975524,-183832
EC00252=-975524,-183832
EC00253=-959628,-183832
EC00254=-832192,-183832
EC00255=-798156,-183832
EC00256=-798156,-183832
EC00257=-798156,-183832
EC00258=-798153,-183835
EC00259=-798156,-183832
EC00260=-798156,-183832
EC00261=-798153,-183835
EC00262=-798156,-183832
EC00263=-798156,-183832
EC00264=-798156,-183832
EC00265=-798156,-183832
EC00266=-798156,-183832
EC00267=-798156,-183832
EC00268=-798156,-183832
EC00269=-798156,-183832
EC00270=-798156,-183832
EC00271=-798156,-183832
EC00272=-798156,-183832
EC00273=-798156,-183832
EC00274=-798156,-183832
EC00275=-798156,-183832
EC00276=-798156,-183832
EC00277=-798156,-183832
EC00278=-798156,-183832
EC00279=-798156,-183832
EC00280=-798156,-183832
EC00281=-798156,-183832
EC00282=-798156,-183832
EC00283=-798156,-183832
EC00284=-798156,-183832
EC00285=-798156,-183832
EC00286=-798156,-183832
EC00287=-798156,-183832
EC00288=-798156,-183832
EC00289=-798156,-183832
EC00290=-798156,-183832
EC00291=-798156,-183832
EC00292=-798156,-183832
EC00293=-798156,-183832
EC00294=-798156,-183832
EC00295=-798156,-183832
EC00296=-798156,-183832
EC00297=-798156,-183832
EC00298=-798156,-183832
EC00299=-798156,-183832
EC00300=-798156,-183832
EC00301=-798156,-183832
EC00302=-798156,-183832
EC00303=-798156,-183832
EC00304=-798156,-183832
EC00305=-798156,-183832
EC00306=-798156,-183832
EC00307=-798156,-183832
EC00308=-798156,-183832
EC00309=-798156,-183832
EC00310=-798156,-183832
EC00311=-798156,-183832
EC00312=-798156,-183832
EC00313=-798156,-183832
EC00314=-798156,-183832
EC00315=-798156,-183832
EC00316=-798156,-183832
EC00317=-798156,-183832
EC00318=-798156,-183832
EC00319=-798156,-183832
EC00320=-798156,-183832
EC00321=-798156,-183832
EC00322=-798156,-183832
EC00323=-798156,-183832
EC00324=-798156,-183832
EC00325=-798156,-183832
EC00326=-798156,-183832
EC00327=-798156,-183832
EC00328=-798156,-183832
EC00329=-798156,-183832
EC00330=-798156,-183832
EC00331=-798156,-183832
EC00332=-798156,-183832
EC00333=-798156,-183832
EC00334=-798156,-183832
EC00335=-798156,-183832
EC00336=-798156,-183832
EC00337=-798156,-183832
EC00338=-798156,-183832
EC00339=-798156,-183832
EC00340=-798156,-183832
EC00341=-798156,-183832
EC00342=-798156,-183832
EC00343=-798156,-183832
EC00344=-798156,-183832
EC00345=-798156,-183832
EC00346=-798156,-183832
EC00347=-798156,-183832
EC00348=-798156,-183832
EC00349=-798155,-183833
EC00350=-798154,-183834
EC00351=-798154,-183834
EC00352=-798154,-183834
EC00353=-798155,-183833
EC00354=-798155,-183833
EC00355=-798156,-183832
EC00356=-798156,-183832
EC00357=-798156,-183832
EC00358=-798155,-183832
EC00359=-798156,-183832
EC00360=-798156,-183832
EC00361=-798156,-183832
EC00362=-798156,-183832
EC00363=-798156,-183832
EC00364=-798156,-183832
EC00365=-798156,-183832
EC00366=-798156,-183832
EC00367=-798156,-183832
EC00368=-798156,-183832
EC00369=-798156,-183832
EC00370=-798156,-183832
EC00371=-798156,-183832
EC00372=-798156,-183832
EC00373=-798156,-183832
EC00374=-798156,-183832
EC00375=-798156,-183832
EC00376=-798156,-183832
EC00377=-798156,-183832
EC00378=-798156,-183832
EC00379=-798156,-183832
EC00380=-798156,-183832
EC00381=-798156,-183832
EC00382=-798156,-183832
EC00383=-798156,-183832
EC00384=-798156,-183832
EC00385=-798156,-183832
EC00386=-798156,-183832
EC00387=-798156,-183832
EC00388=-798156,-183832
EC00389=-798156,-183832
EC00390=-798156,-183832
EC00391=-798156,-183832
EC00392=-798156,-183832
EC00393=-798156,-183832
EC00394=-798156,-183832
EC00395=-798156,-183832
EC00396=-798156,-183832
EC00397=-798156,-183832
EC00398=-798156,-183832
EC00399=-798156,-183832
EC00400=-798156,-183832
EC00401=-798156,-183832
EC00402=-798156,-183832
EC00403=-798156,-183832
EC00404=-798156,-183832
EC00405=-798156,-183832
EC00406=-798156,-183832
EC00407=-798156,-183832
EC00408=-798156,-183832
EC00409=-798156,-183832
EC00410=-798156,-183832
EC00411=-798155,-183832
EC00412=-798156,-183832
EC00413=-798156,-183832
EC00414=-798155,-183832
EC00415=-798156,-183832
EC00416=-798156,-183832
EC00417=-798156,-183832
EC00418=-798156,-183832
EC00419=-798154,-183833
EC00420=-798156,-183832
EC00421=-798156,-183832
EC00422=-798154,-183833
EC00423=-798156,-183832
EC00424=-798156,-183832
EC00425=-798156,-183832
EC00426=-798156,-183832
EC00427=-798156,-183832
EC00428=-798156,-183832
EC00429=-798156,-183832
EC00430=-798156,-183832
EC00431=-798156,-183832
EC00432=-798156,-183832
EC00433=-798156,-183832
EC00434=-798156,-183832
EC00435=-798156,-183832
EC00436=-798156,-183832
EC00437=-798156,-183832
EC00438=-798156,-183832
EC00439=-798156,-183832
EC00440=-798156,-183832
EC00441=-798156,-183832
EC00442=-798156,-183832
EC00443=-798156,-183832
EC00444=-798156,-183832
EC00445=-798156,-183832
EC00446=-798156,-183832
EC00447=-798156,-183832
EC00448=-798156,-183832
EC00449=-798156,-183832
EC00450=-798156,-183832
EC00451=-798156,-183832
EC00452=-798156,-183832
EC00453=-798156,-183832
EC00454=-798156,-183832
///POSTYPE BASE
///RECTAN
///RCONF 0,0,0,0,1,0,0,0,0,0,0,0,0,0,0,0,0,0,0,0,0,0,0,0
P00006=2.006,1.622,-0.565,0.0000,0.0000,0.0000
P00021=0.073,2.058,-0.109,0.0000,0.0000,0.0000
P00022=2.006,1.622,-0.565,0.0000,0.0000,0.0000
///RCONF 0,0,0,0,0,0,0,0,0,0,0,0,0,0,0,0,0,0,0,0,0,0,0,0
P00024=-1.466,-0.226,-0.419,0.0000,0.0000,0.0000
P00025=3.643,0.007,-2.585,0.0000,0.0000,0.0000
P00026=2.644,0.055,-2.583,0.0000,0.0000,0.0000
P00027=2.278,0.099,-4.210,0.0000,0.0000,0.0000
P00032=-0.423,0.157,3.222,0.0000,0.0000,0.0000
P00041=-0.109,0.014,0.966,0.0000,0.0000,0.0000
P00042=-0.220,0.371,-0.613,0.0000,0.0000,0.0000
P00043=-0.179,-5.890,-3.227,0.0000,0.0000,0.0000
P00044=-8.560,-7.557,-5.232,0.0000,0.0000,0.0000
P00045=-8.836,-6.632,-1.438,0.0000,0.0000,0.0000
P00046=-7.725,-0.107,-2.878,0.0000,0.0000,0.0000
P00066=2360.514,789.486,-255.123,0.6232,35.5414,175.8162
P00067=2354.696,158.615,-258.055,26.2211,34.3929,-169.2888
P00068=0.486,-3.949,-12.696,0.0000,0.0000,0.0000
//INST
///DATE 2024/11/20 09:30
///ATTR SC,RW
///GROUP1 RB1,BS1
///GROUP2 ST1
NOP
'OK_r2_O57-69(1)(90,0)
'Down
'Path S1900
SFTOF3D
'Path S1901
SFTOF3D
MOVJ C00000 BC00000 VJ=40.00  +MOVJ EC00000 VJ=15.00
MOVJ C00001 BC00001 VJ=100.00  +MOVJ EC00001 VJ=100.00
MOVL C00002 BC00002 V=400.0  +MOVJ EC00002 VJ=100.00
SMOVL C00003 BC00003 V=100.0  +MOVJ EC00003
SREFP 3 C00004 BC00004  +REFP EC00004
CALL JOB:SEARCH-R1-S13D
SET P026 P006
SFTON3D P026
SMOVL C00005 BC00005 V=100.0  +MOVJ EC00005
SREFP 3 C00006 BC00006  +REFP EC00006
CALL JOB:SEARCH-R1-S13D
SET P026 P006
SFTON3D P026
SMOVL C00007 BC00007 V=100.0  +MOVJ EC00007
MOVL C00008 BC00008 V=400.0  +MOVJ EC00008 VJ=100.00
MOVL C00009 BC00009 V=1000.0  +MOVJ EC00009 VJ=100.00
'Path S1902
SFTOF3D
MOVJ C00010 BC00010 VJ=100.00  +MOVJ EC00010 VJ=100.00
MOVL C00011 BC00011 V=400.0  +MOVJ EC00011 VJ=100.00
SMOVL C00012 BC00012 V=100.0  +MOVJ EC00012
SREFP 3 C00013 BC00013  +REFP EC00013
CALL JOB:SEARCH-R1-S13D
SET P027 P006
SFTON3D P027
SMOVL C00014 BC00014 V=100.0  +MOVJ EC00014
SREFP 3 C00015 BC00015  +REFP EC00015
CALL JOB:SEARCH-R1-S13D
SET P027 P006
SFTON3D P027
SMOVL C00016 BC00016 V=100.0  +MOVJ EC00016
SFTOF3D
MOVL C00017 BC00017 V=400.0  +MOVJ EC00017 VJ=100.00
MOVL C00018 BC00018 V=1000.0  +MOVJ EC00018 VJ=100.00
MOVJ C00019 BC00019 VJ=100.00  +MOVJ EC00019 VJ=100.00
'Path S1903
SFTOF3D
MOVJ C00020 BC00020 VJ=100.00  +MOVJ EC00020 VJ=100.00
MOVL C00021 BC00021 V=400.0  +MOVJ EC00021 VJ=100.00
SMOVL C00022 BC00022 V=100.0  +MOVJ EC00022
SREFP 3 C00023 BC00023  +REFP EC00023
CALL JOB:SEARCH-R1-S13D
SET P022 P006
SFTON3D P022
SMOVL C00024 BC00024 V=100.0  +MOVJ EC00024
SMOVL C00025 BC00025 V=100.0  +MOVJ EC00025
SMOVL C00026 BC00026 V=100.0  +MOVJ EC00026
SREFP 3 C00027 BC00027  +REFP EC00027
CALL JOB:SEARCH-R1-S13D
SET P022 P006
SFTON3D P022
SMOVL C00028 BC00028 V=100.0  +MOVJ EC00028
SFTOF3D
MOVL C00029 BC00029 V=400.0  +MOVJ EC00029 VJ=100.00
SMOVL C00030 BC00030 V=1000.0  +MOVJ EC00030
SMOVL C00031 BC00031 V=1000.0  +MOVJ EC00031
SMOVL C00032 BC00032 V=166.7  +MOVJ EC00032
SREFP 3 C00033 BC00033  +REFP EC00033
CALL JOB:SEARCH-R1-S13D
SET P066 P006
SFTON3D P066
SMOVL C00034 BC00034 V=250.0  +MOVJ EC00034
SMOVL C00035 BC00035 V=250.0  +MOVJ EC00035
SMOVL C00036 BC00036 V=250.0  +MOVJ EC00036
SREFP 3 C00037 BC00037  +REFP EC00037
CALL JOB:SEARCH-R1-S13D
SET P066 P006
SFTON3D P066
SMOVL C00038 BC00038 V=250.0  +MOVJ EC00038
SMOVL C00039 BC00039 V=1000.0  +MOVJ EC00039
SFTOF3D
SMOVL C00040 BC00040 V=1000.0  +MOVJ EC00040
SMOVL C00041 BC00041 V=166.7  +MOVJ EC00041
SREFP 3 C00042 BC00042  +REFP EC00042
CALL JOB:SEARCH-R1-S13D
SET P068 P006
SFTON3D P068
SMOVL C00043 BC00043 V=250.0  +MOVJ EC00043
SREFP 3 C00044 BC00044  +REFP EC00044
CALL JOB:SEARCH-R1-S13D
SET P068 P006
SFTON3D P068
SMOVL C00045 BC00045 V=250.0  +MOVJ EC00045
SMOVL C00046 BC00046 V=166.7  +MOVJ EC00046
SREFP 3 C00047 BC00047  +REFP EC00047
CALL JOB:SEARCH-R1-S13D
SET P068 P006
SFTON3D P068
SMOVL C00048 BC00048 V=250.0  +MOVJ EC00048
SFTOF3D
SMOVL C00049 BC00049 V=1000.0  +MOVJ EC00049
MOVJ C00050 BC00050 VJ=100.00  +MOVJ EC00050 VJ=100.00
MOVJ C00051 BC00051 VJ=100.00  +MOVJ EC00051 VJ=100.00
COMM PAUSE
COMM MOVJ C00052 BC00052 VJ=100.00  +MOVJ EC00052 VJ=100.00
COMM SMOVL C00053 BC00053 V=1000.0  +MOVJ EC00053
COMM SMOVL C00054 BC00054 V=166.7  +MOVJ EC00054
COMM SREFP 3 C00055 BC00055  +REFP EC00055
COMM CALL JOB:SEARCH-R1-S13D
COMM SET P067 P006
COMM SFTON3D P067
COMM SMOVL C00056 BC00056 V=250.0  +MOVJ EC00056
COMM SMOVL C00057 BC00057 V=250.0  +MOVJ EC00057
COMM SMOVL C00058 BC00058 V=133.3  +MOVJ EC00058
COMM SREFP 3 C00059 BC00059  +REFP EC00059
COMM CALL JOB:SEARCH-R1-S13D
COMM SET P067 P006
COMM SFTON3D P067
COMM SMOVL C00060 BC00060 V=250.0  +MOVJ EC00060
COMM SFTOF3D
COMM SMOVL C00061 BC00061 V=1000.0  +MOVJ EC00061
SMOVL C00062 BC00062 V=1000.0  +MOVJ EC00062
MOVJ C00063 BC00063 VJ=100.00  +MOVJ EC00063 VJ=50.00
MOVJ C00064 BC00064 VJ=100.00  +MOVJ EC00064 VJ=100.00
MOVL C00065 BC00065 V=400.0  +MOVJ EC00065 VJ=100.00
SMOVL C00066 BC00066 V=100.0  +MOVJ EC00066
SREFP 3 C00067 BC00067  +REFP EC00067
CALL JOB:SEARCH-R1-S13D
SET P021 P006
SFTON3D P021
SMOVL C00068 BC00068 V=100.0  +MOVJ EC00068
SMOVL C00069 BC00069 V=100.0  +MOVJ EC00069
SREFP 3 C00070 BC00070  +REFP EC00070
CALL JOB:SEARCH-R1-S13D
SET P021 P006
SFTON3D P021
SMOVL C00071 BC00071 V=100.0  +MOVJ EC00071
SMOVL C00072 BC00072 V=100.0  +MOVJ EC00072
SREFP 3 C00073 BC00073  +REFP EC00073
CALL JOB:SEARCH-R1-S13D
SET P021 P006
SFTON3D P021
SMOVL C00074 BC00074 V=100.0  +MOVJ EC00074
MOVL C00075 BC00075 V=400.0  +MOVJ EC00075 VJ=100.00
MOVL C00076 BC00076 V=1000.0  +MOVJ EC00076 VJ=100.00
MOVJ C00077 BC00077 VJ=100.00  +MOVJ EC00077 VJ=100.00
MOVJ C00078 BC00078 VJ=100.00  +MOVJ EC00078 VJ=100.00
MOVJ C00079 BC00079 VJ=100.00  +MOVJ EC00079 VJ=100.00
MOVJ C00080 BC00080 VJ=100.00  +MOVJ EC00080 VJ=100.00
'Path S1912
SFTOF3D
MOVJ C00081 BC00081 VJ=100.00  +MOVJ EC00081 VJ=100.00
MOVL C00082 BC00082 V=400.0  +MOVJ EC00082 VJ=100.00
SMOVL C00083 BC00083 V=100.0  +MOVJ EC00083
SREFP 3 C00084 BC00084  +REFP EC00084
CALL JOB:SEARCH-R1-S13D
SET P032 P006
SFTON3D P032
SMOVL C00085 BC00085 V=100.0  +MOVJ EC00085
SMOVL C00086 BC00086 V=100.0  +MOVJ EC00086
SREFP 3 C00087 BC00087  +REFP EC00087
CALL JOB:SEARCH-R1-S13D
SET P032 P006
SFTON3D P032
SMOVL C00088 BC00088 V=100.0  +MOVJ EC00088
SFTOF3D
MOVL C00089 BC00089 V=400.0  +MOVJ EC00089 VJ=100.00
MOVL C00090 BC00090 V=1000.0  +MOVJ EC00090 VJ=100.00
MOVJ C00091 BC00091 VJ=100.00  +MOVJ EC00091 VJ=100.00
MOVJ C00092 BC00092 VJ=100.00  +MOVJ EC00092 VJ=100.00
'Up
MOVJ C00093 BC00093 VJ=100.00  +MOVJ EC00093 VJ=50.00
MOVJ C00094 BC00094 VJ=100.00  +MOVJ EC00094 VJ=100.00
MOVJ C00095 BC00095 VJ=100.00  +MOVJ EC00095 VJ=100.00
MOVJ C00096 BC00096 VJ=100.00  +MOVJ EC00096 VJ=100.00
MOVJ C00097 BC00097 VJ=100.00  +MOVJ EC00097 VJ=100.00
'Path S1137
SFTOF3D
MOVJ C00098 BC00098 VJ=100.00  +MOVJ EC00098 VJ=100.00
MOVL C00099 BC00099 V=400.0  +MOVJ EC00099 VJ=100.00
SMOVL C00100 BC00100 V=100.0  +MOVJ EC00100
SREFP 3 C00101 BC00101  +REFP EC00101
CALL JOB:SEARCH-R1-S13D
SET P046 P006
SFTON3D P046
SMOVL C00102 BC00102 V=100.0  +MOVJ EC00102
SMOVL C00103 BC00103 V=100.0  +MOVJ EC00103
SREFP 3 C00104 BC00104  +REFP EC00104
CALL JOB:SEARCH-R1-S13D
SET P046 P006
SFTON3D P046
SMOVL C00105 BC00105 V=100.0  +MOVJ EC00105
MOVL C00106 BC00106 V=400.0  +MOVJ EC00106 VJ=100.00
MOVL C00107 BC00107 V=1000.0  +MOVJ EC00107 VJ=100.00
'Path S1169
SFTOF3D
MOVJ C00108 BC00108 VJ=100.00  +MOVJ EC00108 VJ=100.00
MOVL C00109 BC00109 V=400.0  +MOVJ EC00109 VJ=100.00
SMOVL C00110 BC00110 V=100.0  +MOVJ EC00110
SREFP 3 C00111 BC00111  +REFP EC00111
CALL JOB:SEARCH-R1-S13D
SET P045 P006
SFTON3D P045
SMOVL C00112 BC00112 V=100.0  +MOVJ EC00112
SREFP 3 C00113 BC00113  +REFP EC00113
CALL JOB:SEARCH-R1-S13D
SET P045 P006
SFTON3D P045
SMOVL C00114 BC00114 V=100.0  +MOVJ EC00114
SREFP 3 C00115 BC00115  +REFP EC00115
CALL JOB:SEARCH-R1-S13D
SET P045 P006
SFTON3D P045
SMOVL C00116 BC00116 V=100.0  +MOVJ EC00116
SFTOF3D
MOVL C00117 BC00117 V=400.0  +MOVJ EC00117 VJ=100.00
MOVL C00118 BC00118 V=1000.0  +MOVJ EC00118 VJ=100.00
MOVL C00119 BC00119 V=1000.0  +MOVJ EC00119 VJ=100.00
MOVJ C00120 BC00120 VJ=100.00  +MOVJ EC00120 VJ=50.00
MOVJ C00121 BC00121 VJ=100.00  +MOVJ EC00121 VJ=50.00
MOVJ C00122 BC00122 VJ=100.00  +MOVJ EC00122 VJ=100.00
MOVL C00123 BC00123 V=400.0  +MOVJ EC00123 VJ=100.00
SMOVL C00124 BC00124 V=100.0  +MOVJ EC00124
SREFP 3 C00125 BC00125  +REFP EC00125
CALL JOB:SEARCH-R1-S13D
SET P043 P006
SFTON3D P043
SMOVL C00126 BC00126 V=100.0  +MOVJ EC00126
SMOVL C00127 BC00127 V=100.0  +MOVJ EC00127
SREFP 3 C00128 BC00128  +REFP EC00128
CALL JOB:SEARCH-R1-S13D
SET P043 P006
SFTON3D P043
SMOVL C00129 BC00129 V=100.0  +MOVJ EC00129
SMOVL C00130 BC00130 V=100.0  +MOVJ EC00130
SREFP 3 C00131 BC00131  +REFP EC00131
CALL JOB:SEARCH-R1-S13D
SET P043 P006
SFTON3D P043
SMOVL C00132 BC00132 V=100.0  +MOVJ EC00132
MOVL C00133 BC00133 V=400.0  +MOVJ EC00133 VJ=100.00
MOVL C00134 BC00134 V=1000.0  +MOVJ EC00134 VJ=100.00
'Path S1166
SFTOF3D
MOVJ C00135 BC00135 VJ=100.00  +MOVJ EC00135 VJ=100.00
MOVL C00136 BC00136 V=400.0  +MOVJ EC00136 VJ=100.00
SMOVL C00137 BC00137 V=100.0  +MOVJ EC00137
SREFP 3 C00138 BC00138  +REFP EC00138
CALL JOB:SEARCH-R1-S13D
SET P042 P006
SFTON3D P042
SMOVL C00139 BC00139 V=100.0  +MOVJ EC00139
SMOVL C00140 BC00140 V=100.0  +MOVJ EC00140
SREFP 3 C00141 BC00141  +REFP EC00141
CALL JOB:SEARCH-R1-S13D
SET P042 P006
SFTON3D P042
SMOVL C00142 BC00142 V=100.0  +MOVJ EC00142
SMOVL C00143 BC00143 V=100.0  +MOVJ EC00143
SREFP 3 C00144 BC00144  +REFP EC00144
CALL JOB:SEARCH-R1-S13D
SET P042 P006
SFTON3D P042
SMOVL C00145 BC00145 V=100.0  +MOVJ EC00145
MOVL C00146 BC00146 V=400.0  +MOVJ EC00146 VJ=100.00
MOVL C00147 BC00147 V=1000.0  +MOVJ EC00147 VJ=100.00
'Path S1165
SFTOF3D
MOVJ C00148 BC00148 VJ=100.00  +MOVJ EC00148 VJ=100.00
MOVL C00149 BC00149 V=400.0  +MOVJ EC00149 VJ=100.00
SMOVL C00150 BC00150 V=100.0  +MOVJ EC00150
SREFP 3 C00151 BC00151  +REFP EC00151
CALL JOB:SEARCH-R1-S13D
SET P041 P006
SFTON3D P041
SMOVL C00152 BC00152 V=100.0  +MOVJ EC00152
SMOVL C00153 BC00153 V=100.0  +MOVJ EC00153
SREFP 3 C00154 BC00154  +REFP EC00154
CALL JOB:SEARCH-R1-S13D
SET P041 P006
SFTON3D P041
SMOVL C00155 BC00155 V=100.0  +MOVJ EC00155
SMOVL C00156 BC00156 V=100.0  +MOVJ EC00156
SREFP 3 C00157 BC00157  +REFP EC00157
CALL JOB:SEARCH-R1-S13D
SET P041 P006
SFTON3D P041
SMOVL C00158 BC00158 V=100.0  +MOVJ EC00158
MOVL C00159 BC00159 V=400.0  +MOVJ EC00159 VJ=100.00
MOVL C00160 BC00160 V=1000.0  +MOVJ EC00160 VJ=100.00
'Path W378
SFTOF3D
SFTON3D P041
MOVJ C00161 BC00161 VJ=100.00  +MOVJ EC00161 VJ=100.00
SMOVL C00162 BC00162 V=400.0  +MOVJ EC00162
SMOVL C00163 BC00163 V=133.3 PL=0  +MOVJ EC00163
SREFP 1 C00164 BC00164  +REFP EC00164
SREFP 2 C00165 BC00165  +REFP EC00165
MACRO1 MJ#(0) ARGF9
ARCON
SWVON WEV#(61)
SMOVL C00166 BC00166 V=6.7  +MOVJ EC00166
SMOVL C00167 BC00167 V=6.7  +MOVJ EC00167
SMOVL C00168 BC00168 V=6.7  +MOVJ EC00168
ARCOF
SWVOF
SMOVL C00169 BC00169 V=400.0  +MOVJ EC00169
SMOVL C00170 BC00170 V=1000.0  +MOVJ EC00170
SFTOF3D
MOVJ C00171 BC00171 VJ=100.00  +MOVJ EC00171 VJ=100.00
'Path W379
SFTOF3D
SFTON3D P042
MOVJ C00172 BC00172 VJ=100.00  +MOVJ EC00172 VJ=100.00
MOVJ C00173 BC00173 VJ=100.00  +MOVJ EC00173 VJ=100.00
SMOVL C00174 BC00174 V=400.0  +MOVJ EC00174
SMOVL C00175 BC00175 V=133.3 PL=0  +MOVJ EC00175
SREFP 1 C00176 BC00176  +REFP EC00176
SREFP 2 C00177 BC00177  +REFP EC00177
MACRO1 MJ#(0) ARGF9
ARCON
SMOVL C00178 BC00178 V=9.2  +MOVJ EC00178
SMOVL C00179 BC00179 V=9.2  +MOVJ EC00179
SMOVL C00180 BC00180 V=9.2  +MOVJ EC00180
ARCOF
SMOVL C00181 BC00181 V=400.0  +MOVJ EC00181
SMOVL C00182 BC00182 V=1000.0  +MOVJ EC00182
SFTOF3D
MOVJ C00183 BC00183 VJ=20.00  +MOVJ EC00183 VJ=100.00
'Path W380
SFTOF3D
SFTON3D P043
MOVJ C00184 BC00184 VJ=100.00  +MOVJ EC00184 VJ=100.00
MOVJ C00185 BC00185 VJ=100.00  +MOVJ EC00185 VJ=100.00
SMOVL C00186 BC00186 V=400.0  +MOVJ EC00186
SMOVL C00187 BC00187 V=133.3 PL=0  +MOVJ EC00187
SREFP 1 C00188 BC00188  +REFP EC00188
SREFP 2 C00189 BC00189  +REFP EC00189
ARCON
SMOVL C00190 BC00190 V=9.2  +MOVJ EC00190
SMOVL C00191 BC00191 V=9.2  +MOVJ EC00191
ARCOF
SMOVL C00192 BC00192 V=400.0  +MOVJ EC00192
SMOVL C00193 BC00193 V=1000.0  +MOVJ EC00193
SMOVL C00194 BC00194 V=1000.0  +MOVJ EC00194
MOVJ C00195 BC00195 VJ=100.00  +MOVJ EC00195 VJ=100.00
SFTOF3D
'NIE SPAWAMY
COMM 'Path W381
COMM SFTOF3D
COMM SFTON3D P044
COMM MOVJ C00196 BC00196 VJ=100.00  +MOVJ EC00196 VJ=100.00
COMM SMOVL C00197 BC00197 V=400.0  +MOVJ EC00197
COMM SMOVL C00198 BC00198 V=100.0 PL=0  +MOVJ EC00198
COMM SREFP 1 C00199 BC00199  +REFP EC00199
COMM SREFP 2 C00200 BC00200  +REFP EC00200
COMM MACRO1 MJ#(0) ARGF0
COMM ARCON
COMM SMOVL C00201 BC00201 V=10.0  +MOVJ EC00201
COMM SMOVL C00202 BC00202 V=10.0  +MOVJ EC00202
COMM SMOVL C00203 BC00203 V=10.0  +MOVJ EC00203
COMM SMOVL C00204 BC00204 V=10.0  +MOVJ EC00204
COMM SMOVL C00205 BC00205 V=10.0  +MOVJ EC00205
COMM SMOVL C00206 BC00206 V=10.0  +MOVJ EC00206
COMM SMOVL C00207 BC00207 V=10.0  +MOVJ EC00207
COMM SMOVL C00208 BC00208 V=10.0  +MOVJ EC00208
COMM SMOVL C00209 BC00209 V=10.0  +MOVJ EC00209
COMM SMOVL C00210 BC00210 V=10.0  +MOVJ EC00210
COMM SMOVL C00211 BC00211 V=10.0  +MOVJ EC00211
COMM SMOVL C00212 BC00212 V=10.0  +MOVJ EC00212
COMM SMOVL C00213 BC00213 V=10.0  +MOVJ EC00213
COMM SMOVL C00214 BC00214 V=10.0  +MOVJ EC00214
COMM SMOVL C00215 BC00215 V=10.0  +MOVJ EC00215
COMM SMOVL C00216 BC00216 V=10.0  +MOVJ EC00216
COMM SMOVL C00217 BC00217 V=10.0  +MOVJ EC00217
COMM SMOVL C00218 BC00218 V=10.0  +MOVJ EC00218
COMM SMOVL C00219 BC00219 V=10.0  +MOVJ EC00219
COMM SMOVL C00220 BC00220 V=10.0  +MOVJ EC00220
COMM SMOVL C00221 BC00221 V=10.0  +MOVJ EC00221
COMM SMOVL C00222 BC00222 V=10.0  +MOVJ EC00222
COMM SMOVL C00223 BC00223 V=10.0  +MOVJ EC00223
COMM SMOVL C00224 BC00224 V=10.0  +MOVJ EC00224
COMM SMOVL C00225 BC00225 V=10.0  +MOVJ EC00225
COMM ARCOF
COMM SMOVL C00226 BC00226 V=400.0  +MOVJ EC00226
COMM SMOVL C00227 BC00227 V=1000.0  +MOVJ EC00227
COMM SFTOF3D
'Path W382
SFTOF3D
MOVJ C00228 BC00228 VJ=100.00  +MOVJ EC00228 VJ=50.00
SFTON3D P045
MOVJ C00229 BC00229 VJ=100.00  +MOVJ EC00229 VJ=100.00
SMOVL C00230 BC00230 V=400.0  +MOVJ EC00230
SMOVL C00231 BC00231 V=133.3 PL=0  +MOVJ EC00231
SREFP 1 C00232 BC00232  +REFP EC00232
SREFP 2 C00233 BC00233  +REFP EC00233
ARCON
SMOVL C00234 BC00234 V=9.2  +MOVJ EC00234
SMOVL C00235 BC00235 V=9.2  +MOVJ EC00235
SMOVL C00236 BC00236 V=9.2  +MOVJ EC00236
ARCOF
SMOVL C00237 BC00237 V=400.0  +MOVJ EC00237
SMOVL C00238 BC00238 V=1000.0  +MOVJ EC00238
SMOVL C00239 BC00239 V=1000.0  +MOVJ EC00239
SFTOF3D
MOVJ C00240 BC00240 VJ=100.00  +MOVJ EC00240 VJ=100.00
'Path W383
SFTOF3D
SFTON3D P046
MOVJ C00241 BC00241 VJ=100.00  +MOVJ EC00241 VJ=100.00
MOVJ C00242 BC00242 VJ=100.00  +MOVJ EC00242 VJ=100.00
SMOVL C00243 BC00243 V=400.0  +MOVJ EC00243
SMOVL C00244 BC00244 V=133.3 PL=0  +MOVJ EC00244
SREFP 1 C00245 BC00245  +REFP EC00245
SREFP 2 C00246 BC00246  +REFP EC00246
ARCON
SMOVL C00247 BC00247 V=9.2  +MOVJ EC00247
SMOVL C00248 BC00248 V=9.2  +MOVJ EC00248
SMOVL C00249 BC00249 V=9.2  +MOVJ EC00249
ARCOF
SMOVL C00250 BC00250 V=400.0  +MOVJ EC00250
SMOVL C00251 BC00251 V=1000.0  +MOVJ EC00251
SFTOF3D
MOVJ C00252 BC00252 VJ=100.00  +MOVJ EC00252 VJ=100.00
MOVJ C00253 BC00253 VJ=100.00  +MOVJ EC00253 VJ=100.00
'Down
MOVJ C00254 BC00254 VJ=100.00  +MOVJ EC00254 VJ=100.00
MOVJ C00255 BC00255 VJ=100.00  +MOVJ EC00255 VJ=100.00
'Path W1720
SFTOF3D
SFTON3D P032
MOVJ C00256 BC00256 VJ=100.00  +MOVJ EC00256 VJ=100.00
SMOVL C00257 BC00257 V=400.0  +MOVJ EC00257
SMOVL C00258 BC00258 V=133.3  +MOVJ EC00258
SREFP 1 C00259 BC00259  +REFP EC00259
SREFP 2 C00260 BC00260  +REFP EC00260
MACRO1 MJ#(0) ARGF21
ARCON
SWVON WEV#(100)
SMOVC C00261 BC00261 V=9.2  +MOVJ EC00261
SMOVC C00262 BC00262 V=9.2  +MOVJ EC00262
SMOVC C00263 BC00263 V=9.2  +MOVJ EC00263
SMOVC C00264 BC00264 V=9.2  +MOVJ EC00264
SMOVC C00265 BC00265 V=9.2  +MOVJ EC00265
SMOVC C00266 BC00266 V=9.2  +MOVJ EC00266
ARCOF
SWVOF
SMOVL C00267 BC00267 V=400.0  +MOVJ EC00267
SMOVL C00268 BC00268 V=1000.0  +MOVJ EC00268
SFTOF3D
MOVJ C00269 BC00269 VJ=100.00  +MOVJ EC00269 VJ=100.00
MOVJ C00270 BC00270 VJ=100.00  +MOVJ EC00270 VJ=100.00
MOVJ C00271 BC00271 VJ=100.00  +MOVJ EC00271 VJ=100.00
MOVJ C00272 BC00272 VJ=100.00  +MOVJ EC00272 VJ=100.00
MOVJ C00273 BC00273 VJ=100.00  +MOVJ EC00273 VJ=100.00
MOVJ C00274 BC00274 VJ=100.00  +MOVJ EC00274 VJ=100.00
'Path W1626
SFTOF3D
SFTON3D P022
MOVJ C00275 BC00275 VJ=100.00  +MOVJ EC00275 VJ=100.00
SMOVL C00276 BC00276 V=250.0  +MOVJ EC00276
SMOVL C00277 BC00277 V=133.3 PL=0  +MOVJ EC00277
SREFP 1 C00278 BC00278  +REFP EC00278
SREFP 2 C00279 BC00279  +REFP EC00279
MACRO1 MJ#(0) ARGF9
ARCON
SMOVC C00280 BC00280 V=9.2  +MOVJ EC00280
SMOVC C00281 BC00281 V=10.0  +MOVJ EC00281
SMOVC C00282 BC00282 V=10.0  +MOVJ EC00282
SMOVC C00283 BC00283 V=10.0  +MOVJ EC00283
SMOVC C00284 BC00284 V=10.0  +MOVJ EC00284
ARCOF
SMOVL C00285 BC00285 V=400.0  +MOVJ EC00285
SFTOF3D
'Path W1627
SFTOF3D
SFTON3D P022
SMOVL C00286 BC00286 V=100.0 PL=0  +MOVJ EC00286
SREFP 1 C00287 BC00287  +REFP EC00287
SREFP 2 C00288 BC00288  +REFP EC00288
ARCON
SMOVL C00289 BC00289 V=10.0  +MOVJ EC00289
SMOVL C00290 BC00290 V=10.0  +MOVJ EC00290
ARCOF
SMOVL C00291 BC00291 V=400.0  +MOVJ EC00291
SMOVL C00292 BC00292 V=1000.0  +MOVJ EC00292
SFTOF3D
MOVJ C00293 BC00293 VJ=100.00  +MOVJ EC00293 VJ=100.00
MACRO1 MJ#(0) ARGF14
SFTON3D P066
SMOVL C00294 BC00294 V=166.7  +MOVJ EC00294
ARCON
SMOVL C00295 BC00295 V=11.7  +MOVJ EC00295
ARCOF
SMOVL C00296 BC00296 V=333.3  +MOVJ EC00296
SFTOF3D
MOVJ C00297 BC00297 VJ=100.00  +MOVJ EC00297 VJ=100.00
MOVJ C00298 BC00298 VJ=100.00  +MOVJ EC00298 VJ=100.00
SMOVL C00299 BC00299 V=666.7  +MOVJ EC00299
SFTON3D P068
SMOVL C00300 BC00300 V=166.7  +MOVJ EC00300
ARCON
SMOVL C00301 BC00301 V=12.5  +MOVJ EC00301
SMOVL C00302 BC00302 V=10.8  +MOVJ EC00302
SMOVL C00303 BC00303 V=10.8  +MOVJ EC00303
SMOVL C00304 BC00304 V=10.8  +MOVJ EC00304
ARCOF
SMOVL C00305 BC00305 V=166.7  +MOVJ EC00305
SMOVL C00306 BC00306 V=666.7  +MOVJ EC00306
SFTOF3D
MOVJ C00307 BC00307 VJ=50.00  +MOVJ EC00307 VJ=50.00
'
MOVJ C00308 BC00308 VJ=100.00  +MOVJ EC00308 VJ=100.00
MOVJ C00309 BC00309 VJ=100.00  +MOVJ EC00309 VJ=100.00
MOVJ C00310 BC00310 VJ=100.00  +MOVJ EC00310 VJ=100.00
'Path W1911
SFTOF3D
MOVJ C00311 BC00311 VJ=100.00  +MOVJ EC00311 VJ=100.00
SMOVL C00312 BC00312 V=166.7  +MOVJ EC00312
SFTON3D P021
SMOVL C00313 BC00313 V=100.0 PL=0  +MOVJ EC00313
SREFP 1 C00314 BC00314  +REFP EC00314
SREFP 2 C00315 BC00315  +REFP EC00315
MACRO1 MJ#(0) ARGF21
ARCON
SWVON WEV#(100)
SMOVC C00316 BC00316 V=9.2  +MOVJ EC00316
SMOVC C00317 BC00317 V=9.2  +MOVJ EC00317
SMOVC C00318 BC00318 V=9.2  +MOVJ EC00318
SMOVC C00319 BC00319 V=9.2  +MOVJ EC00319
ARCOF
SWVOF
SMOVL C00320 BC00320 V=400.0  +MOVJ EC00320
SMOVL C00321 BC00321 V=1000.0  +MOVJ EC00321
SFTOF3D
MOVJ C00322 BC00322 VJ=100.00  +MOVJ EC00322 VJ=100.00
'
MOVJ C00323 BC00323 VJ=100.00  +MOVJ EC00323 VJ=100.00
MOVJ C00324 BC00324 VJ=100.00  +MOVJ EC00324 VJ=100.00
'NIE SPAWAMY
COMM 'Path W1642
COMM SFTOF3D
COMM SFTON3D P024
COMM MOVJ C00325 BC00325 VJ=100.00  +MOVJ EC00325 VJ=100.00
COMM SMOVL C00326 BC00326 V=400.0  +MOVJ EC00326
COMM SMOVL C00327 BC00327 V=100.0 PL=0  +MOVJ EC00327
COMM SREFP 1 C00328 BC00328  +REFP EC00328
COMM SREFP 2 C00329 BC00329  +REFP EC00329
COMM MACRO1 MJ#(0) ARGF0
COMM ARCON
COMM SMOVL C00330 BC00330 V=10.0  +MOVJ EC00330
COMM ARCOF
COMM SMOVL C00331 BC00331 V=400.0  +MOVJ EC00331
COMM SMOVL C00332 BC00332 V=1000.0  +MOVJ EC00332
COMM SFTOF3D
'NIE SPAWAMY
COMM 'Path W1643
COMM SFTOF3D
COMM SFTON3D P025
COMM MOVJ C00333 BC00333 VJ=100.00  +MOVJ EC00333 VJ=100.00
COMM SMOVL C00334 BC00334 V=400.0  +MOVJ EC00334
COMM SMOVL C00335 BC00335 V=100.0 PL=0  +MOVJ EC00335
COMM SREFP 1 C00336 BC00336  +REFP EC00336
COMM SREFP 2 C00337 BC00337  +REFP EC00337
COMM MACRO1 MJ#(0) ARGF0
COMM ARCON
COMM SMOVL C00338 BC00338 V=10.0  +MOVJ EC00338
COMM ARCOF
COMM SMOVL C00339 BC00339 V=400.0  +MOVJ EC00339
COMM SMOVL C00340 BC00340 V=1000.0  +MOVJ EC00340
COMM SMOVL C00341 BC00341 V=1000.0  +MOVJ EC00341
COMM SFTOF3D
'
'Path W1644
SFTOF3D
SFTON3D P026
MOVJ C00342 BC00342 VJ=100.00  +MOVJ EC00342 VJ=100.00
SMOVL C00343 BC00343 V=333.3  +MOVJ EC00343
SMOVL C00344 BC00344 V=133.3 PL=0  +MOVJ EC00344
SREFP 1 C00345 BC00345  +REFP EC00345
SREFP 2 C00346 BC00346  +REFP EC00346
MACRO1 MJ#(0) ARGF9
ARCON
SMOVL C00347 BC00347 V=6.7  +MOVJ EC00347
SMOVL C00348 BC00348 V=6.7  +MOVJ EC00348
SMOVL C00349 BC00349 V=6.7  +MOVJ EC00349
SMOVL C00350 BC00350 V=5.0  +MOVJ EC00350
SMOVL C00351 BC00351 V=5.0  +MOVJ EC00351
SMOVL C00352 BC00352 V=5.0  +MOVJ EC00352
ARCOF
SMOVL C00353 BC00353 V=133.3  +MOVJ EC00353
SMOVL C00354 BC00354 V=333.3  +MOVJ EC00354
SMOVL C00355 BC00355 V=333.3  +MOVJ EC00355
SFTOF3D
'Path W1645
SFTOF3D
SFTON3D P027
MOVJ C00356 BC00356 VJ=50.00  +MOVJ EC00356 VJ=100.00
SMOVL C00357 BC00357 V=166.7  +MOVJ EC00357
SMOVL C00358 BC00358 V=133.3 PL=0  +MOVJ EC00358
SREFP 1 C00359 BC00359  +REFP EC00359
SREFP 2 C00360 BC00360  +REFP EC00360
MACRO1 MJ#(0) ARGF9
ARCON
SMOVL C00361 BC00361 V=6.7  +MOVJ EC00361
SMOVL C00362 BC00362 V=6.7  +MOVJ EC00362
SMOVL C00363 BC00363 V=6.7  +MOVJ EC00363
ARCON
SMOVL C00364 BC00364 V=6.7  +MOVJ EC00364
SMOVL C00365 BC00365 V=6.7  +MOVJ EC00365
ARCOF
SMOVL C00366 BC00366 V=400.0  +MOVJ EC00366
SMOVL C00367 BC00367 V=1000.0  +MOVJ EC00367
SMOVL C00368 BC00368 V=1000.0  +MOVJ EC00368
SFTOF3D
MOVJ C00369 BC00369 VJ=40.00  +MOVJ EC00369 VJ=100.00
MOVJ C00370 BC00370 VJ=100.00  +MOVJ EC00370 VJ=100.00
COMM 'jakie searche do takicj spoin?
COMM MOVJ C00371 BC00371 VJ=100.00  +MOVJ EC00371 VJ=100.00
COMM 'Path W1646
COMM SFTOF3D
COMM MOVJ C00372 BC00372 VJ=100.00  +MOVJ EC00372 VJ=100.00
COMM MOVL C00373 BC00373 V=400.0  +MOVJ EC00373 VJ=100.00
COMM PAUSE
COMM PAUSE
'USUNAC SPAWANIE ZAMKOW
COMM SFTOF3D
COMM SFTON3D P021
COMM SMOVL C00374 BC00374 V=166.7 PL=0  +MOVJ EC00374
COMM SREFP 1 C00375 BC00375  +REFP EC00375
COMM SREFP 2 C00376 BC00376  +REFP EC00376
COMM MACRO1 MJ#(0) ARGF6
COMM ARCON
COMM SMOVL C00377 BC00377 V=4.2  +MOVJ EC00377
COMM ARCOF
COMM MOVL C00378 BC00378 V=400.0  +MOVJ EC00378 VJ=100.00
COMM MOVL C00379 BC00379 V=1000.0  +MOVJ EC00379 VJ=100.00
COMM MOVL C00380 BC00380 V=333.3  +MOVJ EC00380 VJ=100.00
COMM MOVJ C00381 BC00381 VJ=100.00  +MOVJ EC00381 VJ=100.00
COMM 'brak dostÄpu do jednej spoiny
COMM 'Path W1647
COMM SFTOF3D
COMM MOVJ C00382 BC00382 VJ=25.00  +MOVJ EC00382 VJ=100.00
COMM MOVJ C00383 BC00383 VJ=25.00  +MOVJ EC00383 VJ=100.00
COMM MOVL C00384 BC00384 V=400.0  +MOVJ EC00384 VJ=100.00
COMM SFTOF3D
COMM SMOVL C00385 BC00385 V=166.7 PL=0  +MOVJ EC00385
COMM SREFP 1 C00386 BC00386  +REFP EC00386
COMM SREFP 2 C00387 BC00387  +REFP EC00387
COMM MACRO1 MJ#(0) ARGF6
COMM ARCON
COMM SMOVL C00388 BC00388 V=4.2  +MOVJ EC00388
COMM ARCOF
COMM MOVL C00389 BC00389 V=400.0  +MOVJ EC00389 VJ=100.00
COMM MOVL C00390 BC00390 V=1000.0  +MOVJ EC00390 VJ=100.00
COMM 'Path W1648
COMM SFTOF3D
COMM MOVJ C00391 BC00391 VJ=10.00  +MOVJ EC00391 VJ=100.00
COMM MOVL C00392 BC00392 V=166.7  +MOVJ EC00392 VJ=100.00
COMM SFTON3D P021
COMM SMOVL C00393 BC00393 V=100.0 PL=0  +MOVJ EC00393
COMM SREFP 1 C00394 BC00394  +REFP EC00394
COMM SREFP 2 C00395 BC00395  +REFP EC00395
COMM MACRO1 MJ#(0) ARGF6
COMM ARCON
COMM SMOVL C00396 BC00396 V=4.2  +MOVJ EC00396
COMM ARCOF
COMM MOVL C00397 BC00397 V=400.0  +MOVJ EC00397 VJ=100.00
COMM MOVL C00398 BC00398 V=1000.0  +MOVJ EC00398 VJ=100.00
COMM MOVL C00399 BC00399 V=1000.0  +MOVJ EC00399 VJ=100.00
COMM MOVJ C00400 BC00400 VJ=10.00  +MOVJ EC00400 VJ=100.00
COMM 'Path W1649
COMM SFTOF3D
COMM MOVJ C00401 BC00401 VJ=15.00  +MOVJ EC00401 VJ=100.00
COMM MOVL C00402 BC00402 V=166.7  +MOVJ EC00402 VJ=100.00
COMM SFTON3D P021
COMM SMOVL C00403 BC00403 V=166.7 PL=0  +MOVJ EC00403
COMM SREFP 1 C00404 BC00404  +REFP EC00404
COMM SREFP 2 C00405 BC00405  +REFP EC00405
COMM MACRO1 MJ#(0) ARGF6
COMM ARCON
COMM SMOVL C00406 BC00406 V=4.2  +MOVJ EC00406
COMM ARCOF
COMM MOVL C00407 BC00407 V=400.0  +MOVJ EC00407 VJ=100.00
COMM MOVL C00408 BC00408 V=1000.0  +MOVJ EC00408 VJ=100.00
COMM 'Path W1650
COMM MOVJ C00409 BC00409 VJ=100.00  +MOVJ EC00409 VJ=100.00
COMM MOVL C00410 BC00410 V=166.7  +MOVJ EC00410 VJ=100.00
COMM SMOVL C00411 BC00411 V=166.7 PL=0  +MOVJ EC00411
COMM SREFP 1 C00412 BC00412  +REFP EC00412
COMM SREFP 2 C00413 BC00413  +REFP EC00413
COMM MACRO1 MJ#(0) ARGF6
COMM ARCON
COMM SMOVL C00414 BC00414 V=4.2  +MOVJ EC00414
COMM ARCOF
COMM MOVL C00415 BC00415 V=400.0  +MOVJ EC00415 VJ=100.00
COMM MOVL C00416 BC00416 V=1000.0  +MOVJ EC00416 VJ=100.00
COMM 'Path W1651
COMM SFTOF3D
COMM MOVJ C00417 BC00417 VJ=100.00  +MOVJ EC00417 VJ=100.00
COMM MOVL C00418 BC00418 V=400.0  +MOVJ EC00418 VJ=100.00
COMM SFTON3D P021
COMM SMOVL C00419 BC00419 V=166.7 PL=0  +MOVJ EC00419
COMM SREFP 1 C00420 BC00420  +REFP EC00420
COMM SREFP 2 C00421 BC00421  +REFP EC00421
COMM MACRO1 MJ#(0) ARGF6
COMM ARCON
COMM SMOVL C00422 BC00422 V=4.2  +MOVJ EC00422
COMM ARCOF
COMM MOVL C00423 BC00423 V=400.0  +MOVJ EC00423 VJ=100.00
COMM MOVL C00424 BC00424 V=1000.0  +MOVJ EC00424 VJ=100.00
COMM 'Path W1652
COMM SFTOF3D
COMM MOVJ C00425 BC00425 VJ=100.00  +MOVJ EC00425 VJ=100.00
COMM MOVL C00426 BC00426 V=166.7  +MOVJ EC00426 VJ=100.00
COMM SFTON3D P021
COMM SMOVL C00427 BC00427 V=166.7 PL=0  +MOVJ EC00427
COMM SREFP 1 C00428 BC00428  +REFP EC00428
COMM SREFP 2 C00429 BC00429  +REFP EC00429
COMM MACRO1 MJ#(0) ARGF6
COMM ARCON
COMM SMOVL C00430 BC00430 V=4.2  +MOVJ EC00430
COMM ARCOF
COMM MOVL C00431 BC00431 V=166.7  +MOVJ EC00431 VJ=100.00
COMM MOVL C00432 BC00432 V=166.7  +MOVJ EC00432 VJ=100.00
COMM MOVJ C00433 BC00433 VJ=50.00  +MOVJ EC00433 VJ=20.00
COMM SMOVL C00434 BC00434 V=166.7  +MOVJ EC00434
COMM ARCON
COMM SMOVL C00435 BC00435 V=4.2  +MOVJ EC00435
COMM ARCOF
COMM SMOVL C00436 BC00436 V=166.7  +MOVJ EC00436
COMM 'jakie searche do takicj spoin?
COMM MOVJ C00437 BC00437 VJ=100.00  +MOVJ EC00437 VJ=100.00
COMM MOVJ C00438 BC00438 VJ=20.00  +MOVJ EC00438 VJ=100.00
COMM MOVJ C00439 BC00439 VJ=100.00  +MOVJ EC00439 VJ=100.00
COMM MOVJ C00440 BC00440 VJ=100.00  +MOVJ EC00440 VJ=100.00
COMM 'Path W1653
COMM SFTOF3D
COMM MOVJ C00441 BC00441 VJ=100.00  +MOVJ EC00441 VJ=100.00
COMM MOVL C00442 BC00442 V=166.7  +MOVJ EC00442 VJ=100.00
COMM SFTON3D P067
COMM SMOVL C00443 BC00443 V=166.7 PL=0  +MOVJ EC00443
COMM SREFP 1 C00444 BC00444  +REFP EC00444
COMM SREFP 2 C00445 BC00445  +REFP EC00445
COMM ARCON
COMM MACRO1 MJ#(0) ARGF9
COMM SMOVL C00446 BC00446 V=10.8  +MOVJ EC00446
COMM ARCOF
COMM SMOVL C00447 BC00447 V=166.7  +MOVJ EC00447
COMM SMOVL C00448 BC00448 V=666.7  +MOVJ EC00448
COMM SMOVL C00449 BC00449 V=166.7  +MOVJ EC00449
COMM ARCON
COMM SMOVL C00450 BC00450 V=10.8  +MOVJ EC00450
COMM ARCOF
COMM SMOVL C00451 BC00451 V=250.0  +MOVJ EC00451
COMM 'Path W1654
COMM SFTOF3D
COMM MOVJ C00452 BC00452 VJ=100.00  +MOVJ EC00452 VJ=100.00
COMM MOVJ C00453 BC00453 VJ=100.00  +MOVJ EC00453 VJ=100.00
MOVJ C00454 BC00454 VJ=100.00  +MOVJ EC00454 VJ=100.00
'Down
END
